LIN {X 0,Y 358.84,Z 342.917,A -85,B 0,C 180,E1 -13392.769,E2 -13392.769} C_VEL
LIN {X 0,Y 357.605,Z 354.158,A -85,B 0,C 180,E1 -13394.029,E2 -13394.029} C_VEL
LIN {X 0,Y 356.532,Z 364.122,A -85,B 0,C 180,E1 -13395.444,E2 -13395.444} C_VEL
LIN {X 0,Y 355.516,Z 373.786,A -85,B 0,C 180,E1 -13397.15,E2 -13397.15} C_VEL
LIN {X 0,Y 354.57,Z 381.475,A -85,B 0,C 180,E1 -13398.857,E2 -13398.857} C_VEL
LIN {X 0,Y 353.885,Z 388.571,A -85,B 0,C 180,E1 -13400.858,E2 -13400.858} C_VEL
LIN {X 0,Y 353.515,Z 393.294,A -85,B 0,C 180,E1 -13402.575,E2 -13402.575} C_VEL
LIN {X 0,Y 353.31,Z 396.903,A -85,B 0,C 180,E1 -13404.292,E2 -13404.292} C_VEL
LIN {X 0,Y 353.278,Z 398.766,A -85,B 0,C 180,E1 -13405.436,E2 -13405.436} C_VEL
LIN {X 0,Y 353.222,Z 400.162,A -85,B 0,C 180,E1 -13406.578,E2 -13406.578} C_VEL
LIN {X 0,Y 353.216,Z 401.767,A -85,B 0,C 180,E1 -13408.86,E2 -13408.86} C_VEL
LIN {X 0,Y 353.262,Z 401.983,A -85,B 0,C 180,E1 -13410,E2 -13410} C_VEL
LIN {X 0,Y 353.216,Z 401.762,A -85,B 0,C 180,E1 -13411.14,E2 -13411.14} C_VEL
LIN {X 0,Y 353.219,Z 400.153,A -85,B 0,C 180,E1 -13413.422,E2 -13413.422} C_VEL
LIN {X 0,Y 353.263,Z 398.752,A -85,B 0,C 180,E1 -13414.564,E2 -13414.564} C_VEL
LIN {X 0,Y 353.278,Z 396.508,A -85,B 0,C 180,E1 -13415.908,E2 -13415.908} C_VEL
LIN {X 0,Y 353.615,Z 391.828,A -85,B 0,C 180,E1 -13417.997,E2 -13417.997} C_VEL
LIN {X 0,Y 354.162,Z 385.708,A -85,B 0,C 180,E1 -13419.999,E2 -13419.999} C_VEL
LIN {X 0,Y 354.828,Z 379.025,A -85,B 0,C 180,E1 -13421.714,E2 -13421.714} C_VEL
LIN {X 0,Y 355.87,Z 370.739,A -85,B 0,C 180,E1 -13423.418,E2 -13423.418} C_VEL
LIN {X 0,Y 356.797,Z 362.241,A -85,B 0,C 180,E1 -13424.837,E2 -13424.837} C_VEL
LIN {X 0,Y 357.874,Z 351.742,A -85,B 0,C 180,E1 -13426.251,E2 -13426.251} C_VEL
LIN {X 0,Y 359.111,Z 339.929,A -85,B 0,C 180,E1 -13427.511,E2 -13427.511} C_VEL
LIN {X 0,Y 359.835,Z 331.742,A -85,B 0,C 180,E1 -13428.21,E2 -13428.21} C_VEL
LIN {X 0,Y 358.663,Z 320.559,A -85,B 0,C 180,E1 -13429.087,E2 -13429.087} C_VEL
LIN {X 0,Y 356.717,Z 308.163,A -85,B 0,C 180,E1 -13429.872,E2 -13429.872} C_VEL
LIN {X 0,Y 354.087,Z 295.342,A -85,B 0,C 180,E1 -13430.496,E2 -13430.496} C_VEL
LIN {X 0,Y 354.506,Z 288.95,A -85,B 0,C 180,E1 -13434.225,E2 -13434.225} C_VEL
LIN {X 0,Y 355.003,Z 283.001,A -85,B 0,C 180,E1 -13437.725,E2 -13437.725} C_VEL
LIN {X 0,Y 355.574,Z 277.671,A -85,B 0,C 180,E1 -13440.924,E2 -13440.924} C_VEL
LIN {X 0,Y 356.224,Z 271.24,A -85,B 0,C 180,E1 -13444.9,E2 -13444.9} C_VEL
LIN {X 0,Y 356.056,Z 266.77,A -85,B 0,C 180,E1 -13447.857,E2 -13447.857} C_VEL
LIN {X 0,Y 355.303,Z 261.976,A -85,B 0,C 180,E1 -13451.266,E2 -13451.266} C_VEL
LIN {X 0,Y 354.831,Z 259.291,A -85,B 0,C 180,E1 -13453.339,E2 -13453.339} C_VEL
LIN {X 0,Y 354.786,Z 259.29,A -85,B 0,C 180,E1 -13457.133,E2 -13457.133} C_VEL
LIN {X 0,Y 354.785,Z 259.294,A -85,B 0,C 180,E1 -13460.662,E2 -13460.662} C_VEL
LIN {X 0,Y 354.822,Z 259.288,A -85,B 0,C 180,E1 -13464.301,E2 -13464.301} C_VEL
LIN {X 0,Y 354.788,Z 259.289,A -85,B 0,C 180,E1 -13467.667,E2 -13467.667} C_VEL
LIN {X 0,Y 354.802,Z 259.287,A -85,B 0,C 180,E1 -13471.615,E2 -13471.615} C_VEL
LIN {X 0,Y 354.806,Z 259.286,A -85,B 0,C 180,E1 -13475.42,E2 -13475.42} C_VEL
LIN {X 0,Y 354.828,Z 259.283,A -85,B 0,C 180,E1 -13479.113,E2 -13479.113} C_VEL
LIN {X 0,Y 354.9,Z 259.274,A -85,B 0,C 180,E1 -13482.72,E2 -13482.72} C_VEL
LIN {X 0,Y 354.953,Z 259.269,A -85,B 0,C 180,E1 -13486.255,E2 -13486.255} C_VEL
LIN {X 0,Y 354.956,Z 259.271,A -85,B 0,C 180,E1 -13489.735,E2 -13489.735} C_VEL
LIN {X 0,Y 355.113,Z 259.25,A -85,B 0,C 180,E1 -13493.18,E2 -13493.18} C_VEL
LIN {X 0,Y 355.245,Z 259.233,A -85,B 0,C 180,E1 -13497.732,E2 -13497.732} C_VEL
LIN {X 0,Y 355.353,Z 259.218,A -85,B 0,C 180,E1 -13500,E2 -13500} C_VEL
LIN {X 0,Y 355.232,Z 259.233,A -85,B 0,C 180,E1 -13502.268,E2 -13502.268} C_VEL
LIN {X 0,Y 355.107,Z 259.252,A -85,B 0,C 180,E1 -13506.82,E2 -13506.82} C_VEL
LIN {X 0,Y 354.958,Z 259.268,A -85,B 0,C 180,E1 -13510.265,E2 -13510.265} C_VEL
LIN {X 0,Y 354.944,Z 259.269,A -85,B 0,C 180,E1 -13514.019,E2 -13514.019} C_VEL
LIN {X 0,Y 354.891,Z 259.276,A -85,B 0,C 180,E1 -13518.092,E2 -13518.092} C_VEL
LIN {X 0,Y 354.817,Z 259.287,A -85,B 0,C 180,E1 -13522.107,E2 -13522.107} C_VEL
LIN {X 0,Y 354.9,Z 259.275,A -85,B 0,C 180,E1 -13525.828,E2 -13525.828} C_VEL
LIN {X 0,Y 354.855,Z 259.281,A -85,B 0,C 180,E1 -13529.679,E2 -13529.679} C_VEL
LIN {X 0,Y 354.807,Z 259.288,A -85,B 0,C 180,E1 -13533.702,E2 -13533.702} C_VEL
LIN {X 0,Y 354.796,Z 259.289,A -85,B 0,C 180,E1 -13536.46,E2 -13536.46} C_VEL
LIN {X 0,Y 354.825,Z 259.285,A -85,B 0,C 180,E1 -13539.424,E2 -13539.424} C_VEL
LIN {X 0,Y 354.787,Z 259.288,A -85,B 0,C 180,E1 -13542.867,E2 -13542.867} C_VEL
LIN {X 0,Y 354.763,Z 259.293,A -85,B 0,C 180,E1 -13546.103,E2 -13546.103} C_VEL
LIN {X 0,Y 354.763,Z 259.294,A -85,B 0,C 180,E1 -13549.176,E2 -13549.176} C_VEL
LIN {X 0,Y 354.781,Z 259.293,A -85,B 0,C 180,E1 -13552.408,E2 -13552.408} C_VEL
LIN {X 0,Y 354.752,Z 259.395,A -85,B 0,C 180,E1 -13553.535,E2 -13553.535} C_VEL
LIN {X 0,Y 354.712,Z 262.351,A -85,B 0,C 180,E1 -13556.321,E2 -13556.321} C_VEL
LIN {X 0,Y 354.545,Z 265.242,A -85,B 0,C 180,E1 -13558.977,E2 -13558.977} C_VEL
LIN {X 0,Y 354.359,Z 268.174,A -85,B 0,C 180,E1 -13561.576,E2 -13561.576} C_VEL
LIN {X 0,Y 354.181,Z 271.128,A -85,B 0,C 180,E1 -13564.116,E2 -13564.116} C_VEL
LIN {X 0,Y 354.025,Z 274.086,A -85,B 0,C 180,E1 -13566.607,E2 -13566.607} C_VEL
LIN {X 0,Y 353.896,Z 277.951,A -85,B 0,C 180,E1 -13569.582,E2 -13569.582} C_VEL
LIN {X 0,Y 357.36,Z 291.296,A -85,B 0,C 180,E1 -13570.311,E2 -13570.311} C_VEL
LIN {X 0,Y 360.034,Z 303.79,A -85,B 0,C 180,E1 -13571.188,E2 -13571.188} C_VEL
LIN {X 0,Y 360.75,Z 309.963,A -85,B 0,C 180,E1 -13571.676,E2 -13571.676} C_VEL
LIN {X 0,Y 359.733,Z 321.615,A -85,B 0,C 180,E1 -13572.666,E2 -13572.666} C_VEL
LIN {X 0,Y 358.763,Z 332.231,A -85,B 0,C 180,E1 -13573.817,E2 -13573.817} C_VEL
LIN {X 0,Y 357.607,Z 342.508,A -85,B 0,C 180,E1 -13575.198,E2 -13575.198} C_VEL
LIN {X 0,Y 356.595,Z 351.002,A -85,B 0,C 180,E1 -13576.61,E2 -13576.61} C_VEL
LIN {X 0,Y 355.567,Z 359.255,A -85,B 0,C 180,E1 -13578.311,E2 -13578.311} C_VEL
LIN {X 0,Y 354.765,Z 365.902,A -85,B 0,C 180,E1 -13580.018,E2 -13580.018} C_VEL
LIN {X 0,Y 354.082,Z 371.99,A -85,B 0,C 180,E1 -13582.014,E2 -13582.014} C_VEL
LIN {X 0,Y 353.808,Z 375.059,A -85,B 0,C 180,E1 -13583.314,E2 -13583.314} C_VEL
LIN {X 0,Y 353.494,Z 378.859,A -85,B 0,C 180,E1 -13585.439,E2 -13585.439} C_VEL
LIN {X 0,Y 353.335,Z 380.259,A -85,B 0,C 180,E1 -13586.579,E2 -13586.579} C_VEL
LIN {X 0,Y 353.256,Z 381.864,A -85,B 0,C 180,E1 -13588.86,E2 -13588.86} C_VEL
LIN {X 0,Y 353.265,Z 382.096,A -85,B 0,C 180,E1 -13590,E2 -13590} C_VEL
LIN {X 0,Y 353.256,Z 381.907,A -85,B 0,C 180,E1 -13591.14,E2 -13591.14} C_VEL
LIN {X 0,Y 353.332,Z 380.356,A -85,B 0,C 180,E1 -13593.421,E2 -13593.421} C_VEL
LIN {X 0,Y 353.486,Z 378.999,A -85,B 0,C 180,E1 -13594.562,E2 -13594.562} C_VEL
LIN {X 0,Y 353.738,Z 376.181,A -85,B 0,C 180,E1 -13596.247,E2 -13596.247} C_VEL
LIN {X 0,Y 354.088,Z 372.247,A -85,B 0,C 180,E1 -13597.986,E2 -13597.986} C_VEL
LIN {X 0,Y 354.62,Z 367.232,A -85,B 0,C 180,E1 -13599.698,E2 -13599.698} C_VEL
LIN {X 0,Y 355.366,Z 360.917,A -85,B 0,C 180,E1 -13601.407,E2 -13601.407} C_VEL
LIN {X 0,Y 356.347,Z 353.01,A -85,B 0,C 180,E1 -13603.109,E2 -13603.109} C_VEL
LIN {X 0,Y 357.578,Z 343.172,A -85,B 0,C 180,E1 -13604.804,E2 -13604.804} C_VEL
LIN {X 0,Y 358.681,Z 332.659,A -85,B 0,C 180,E1 -13606.237,E2 -13606.237} C_VEL
LIN {X 0,Y 359.616,Z 322.621,A -85,B 0,C 180,E1 -13607.34,E2 -13607.34} C_VEL
LIN {X 0,Y 360.748,Z 310.987,A -85,B 0,C 180,E1 -13608.346,E2 -13608.346} C_VEL
LIN {X 0,Y 360.615,Z 307.38,A -85,B 0,C 180,E1 -13608.628,E2 -13608.628} C_VEL
LIN {X 0,Y 358.493,Z 296.304,A -85,B 0,C 180,E1 -13609.468,E2 -13609.468} C_VEL
LIN {X 0,Y 355.47,Z 283.821,A -85,B 0,C 180,E1 -13610.233,E2 -13610.233} C_VEL
LIN {X 0,Y 353.884,Z 277.728,A -85,B 0,C 180,E1 -13610.556,E2 -13610.556} C_VEL
LIN {X 0,Y 354.106,Z 272.742,A -85,B 0,C 180,E1 -13614.632,E2 -13614.632} C_VEL
LIN {X 0,Y 354.281,Z 269.783,A -85,B 0,C 180,E1 -13617.146,E2 -13617.146} C_VEL
LIN {X 0,Y 354.421,Z 266.827,A -85,B 0,C 180,E1 -13619.719,E2 -13619.719} C_VEL
LIN {X 0,Y 354.596,Z 263.203,A -85,B 0,C 180,E1 -13622.991,E2 -13622.991} C_VEL
LIN {X 0,Y 354.759,Z 260.333,A -85,B 0,C 180,E1 -13625.685,E2 -13625.685} C_VEL
LIN {X 0,Y 354.736,Z 259.52,A -85,B 0,C 180,E1 -13626.467,E2 -13626.467} C_VEL
LIN {X 0,Y 354.774,Z 259.292,A -85,B 0,C 180,E1 -13627.861,E2 -13627.861} C_VEL
LIN {X 0,Y 354.124,Z 259.375,A -85,B 0,C 180,E1 -13628.807,E2 -13628.807} C_VEL
LIN {X 0,Y 351.253,Z 259.732,A -85,B 0,C 180,E1 -13630.347,E2 -13630.347} C_VEL
LIN {X 0,Y 348.817,Z 260.031,A -85,B 0,C 180,E1 -13631.593,E2 -13631.593} C_VEL
LIN {X 0,Y 347.784,Z 260.165,A -85,B 0,C 180,E1 -13632.557,E2 -13632.557} C_VEL
LIN {X 0,Y 347.707,Z 260.167,A -85,B 0,C 180,E1 -13632.884,E2 -13632.884} C_VEL
LIN {X 0,Y 347.727,Z 260.17,A -85,B 0,C 180,E1 -13636.686,E2 -13636.686} C_VEL
LIN {X 0,Y 347.748,Z 260.171,A -85,B 0,C 180,E1 -13640.173,E2 -13640.173} C_VEL
LIN {X 0,Y 347.763,Z 260.164,A -85,B 0,C 180,E1 -13642.679,E2 -13642.679} C_VEL
LIN {X 0,Y 347.751,Z 260.17,A -85,B 0,C 180,E1 -13645.956,E2 -13645.956} C_VEL
LIN {X 0,Y 347.766,Z 260.166,A -85,B 0,C 180,E1 -13649.654,E2 -13649.654} C_VEL
LIN {X 0,Y 347.854,Z 260.151,A -85,B 0,C 180,E1 -13652.745,E2 -13652.745} C_VEL
LIN {X 0,Y 347.787,Z 260.161,A -85,B 0,C 180,E1 -13656.162,E2 -13656.162} C_VEL
LIN {X 0,Y 347.802,Z 260.16,A -85,B 0,C 180,E1 -13659.909,E2 -13659.909} C_VEL
LIN {X 0,Y 347.834,Z 260.158,A -85,B 0,C 180,E1 -13663.568,E2 -13663.568} C_VEL
LIN {X 0,Y 347.893,Z 260.152,A -85,B 0,C 180,E1 -13667.161,E2 -13667.161} C_VEL
LIN {X 0,Y 347.938,Z 260.143,A -85,B 0,C 180,E1 -13670.701,E2 -13670.701} C_VEL
LIN {X 0,Y 348.076,Z 260.13,A -85,B 0,C 180,E1 -13673.042,E2 -13673.042} C_VEL
LIN {X 0,Y 348.195,Z 260.109,A -85,B 0,C 180,E1 -13677.686,E2 -13677.686} C_VEL
LIN {X 0,Y 348.148,Z 260.117,A -85,B 0,C 180,E1 -13681.157,E2 -13681.157} C_VEL
LIN {X 0,Y 348.209,Z 260.11,A -85,B 0,C 180,E1 -13682.313,E2 -13682.313} C_VEL
LIN {X 0,Y 348.08,Z 260.126,A -85,B 0,C 180,E1 -13686.958,E2 -13686.958} C_VEL
LIN {X 0,Y 347.894,Z 260.152,A -85,B 0,C 180,E1 -13690.475,E2 -13690.475} C_VEL
LIN {X 0,Y 347.901,Z 260.15,A -85,B 0,C 180,E1 -13694.15,E2 -13694.15} C_VEL
LIN {X 0,Y 347.894,Z 260.151,A -85,B 0,C 180,E1 -13698.29,E2 -13698.29} C_VEL
LIN {X 0,Y 347.769,Z 260.164,A -85,B 0,C 180,E1 -13701.626,E2 -13701.626} C_VEL
LIN {X 0,Y 347.743,Z 260.166,A -85,B 0,C 180,E1 -13705.114,E2 -13705.114} C_VEL
LIN {X 0,Y 347.74,Z 260.17,A -85,B 0,C 180,E1 -13707.7,E2 -13707.7} C_VEL
LIN {X 0,Y 347.743,Z 260.167,A -85,B 0,C 180,E1 -13710.349,E2 -13710.349} C_VEL
LIN {X 0,Y 347.75,Z 260.167,A -85,B 0,C 180,E1 -13714.044,E2 -13714.044} C_VEL
LIN {X 0,Y 347.758,Z 260.168,A -85,B 0,C 180,E1 -13717.321,E2 -13717.321} C_VEL
LIN {X 0,Y 347.742,Z 260.169,A -85,B 0,C 180,E1 -13721.601,E2 -13721.601} C_VEL
LIN {X 0,Y 347.707,Z 260.175,A -85,B 0,C 180,E1 -13725.027,E2 -13725.027} C_VEL
LIN {X 0,Y 347.797,Z 260.363,A -85,B 0,C 180,E1 -13726.503,E2 -13726.503} C_VEL
LIN {X 0,Y 348.598,Z 264.999,A -85,B 0,C 180,E1 -13730.006,E2 -13730.006} C_VEL
LIN {X 0,Y 349.207,Z 269.003,A -85,B 0,C 180,E1 -13732.859,E2 -13732.859} C_VEL
LIN {X 0,Y 349.145,Z 273.279,A -85,B 0,C 180,E1 -13735.693,E2 -13735.693} C_VEL
LIN {X 0,Y 348.401,Z 279.687,A -85,B 0,C 180,E1 -13739.715,E2 -13739.715} C_VEL
LIN {X 0,Y 347.715,Z 286.034,A -85,B 0,C 180,E1 -13743.598,E2 -13743.598} C_VEL
LIN {X 0,Y 347.277,Z 292.338,A -85,B 0,C 180,E1 -13747.386,E2 -13747.386} C_VEL
LIN {X 0,Y 347.056,Z 295.141,A -85,B 0,C 180,E1 -13749.05,E2 -13749.05} C_VEL
LIN {X 0,Y 350.069,Z 309.551,A -85,B 0,C 180,E1 -13749.797,E2 -13749.797} C_VEL
LIN {X 0,Y 351.916,Z 321.47,A -85,B 0,C 180,E1 -13750.592,E2 -13750.592} C_VEL
LIN {X 0,Y 353.017,Z 333.482,A -85,B 0,C 180,E1 -13751.576,E2 -13751.576} C_VEL
LIN {X 0,Y 351.882,Z 344.141,A -85,B 0,C 180,E1 -13752.567,E2 -13752.567} C_VEL
LIN {X 0,Y 350.633,Z 355.073,A -85,B 0,C 180,E1 -13753.858,E2 -13753.858} C_VEL
LIN {X 0,Y 349.631,Z 363.923,A -85,B 0,C 180,E1 -13755.15,E2 -13755.15} C_VEL
LIN {X 0,Y 348.555,Z 373.587,A -85,B 0,C 180,E1 -13756.889,E2 -13756.889} C_VEL
LIN {X 0,Y 347.55,Z 381.275,A -85,B 0,C 180,E1 -13758.629,E2 -13758.629} C_VEL
LIN {X 0,Y 346.857,Z 388.372,A -85,B 0,C 180,E1 -13760.671,E2 -13760.671} C_VEL
LIN {X 0,Y 346.465,Z 393.095,A -85,B 0,C 180,E1 -13762.423,E2 -13762.423} C_VEL
LIN {X 0,Y 346.23,Z 396.704,A -85,B 0,C 180,E1 -13764.175,E2 -13764.175} C_VEL
LIN {X 0,Y 346.176,Z 398.566,A -85,B 0,C 180,E1 -13765.342,E2 -13765.342} C_VEL
LIN {X 0,Y 346.146,Z 399.963,A -85,B 0,C 180,E1 -13766.508,E2 -13766.508} C_VEL
LIN {X 0,Y 346.116,Z 401.567,A -85,B 0,C 180,E1 -13768.836,E2 -13768.836} C_VEL
LIN {X 0,Y 346.164,Z 401.783,A -85,B 0,C 180,E1 -13770,E2 -13770} C_VEL
LIN {X 0,Y 346.116,Z 401.562,A -85,B 0,C 180,E1 -13771.163,E2 -13771.163} C_VEL
LIN {X 0,Y 346.142,Z 399.953,A -85,B 0,C 180,E1 -13773.492,E2 -13773.492} C_VEL
LIN {X 0,Y 346.16,Z 398.551,A -85,B 0,C 180,E1 -13774.658,E2 -13774.658} C_VEL
LIN {X 0,Y 346.241,Z 395.608,A -85,B 0,C 180,E1 -13776.409,E2 -13776.409} C_VEL
LIN {X 0,Y 346.555,Z 391.626,A -85,B 0,C 180,E1 -13778.161,E2 -13778.161} C_VEL
LIN {X 0,Y 347.136,Z 385.506,A -85,B 0,C 180,E1 -13780.204,E2 -13780.204} C_VEL
LIN {X 0,Y 347.825,Z 378.821,A -85,B 0,C 180,E1 -13781.953,E2 -13781.953} C_VEL
LIN {X 0,Y 348.941,Z 370.536,A -85,B 0,C 180,E1 -13783.689,E2 -13783.689} C_VEL
LIN {X 0,Y 350.023,Z 360.981,A -85,B 0,C 180,E1 -13785.292,E2 -13785.292} C_VEL
LIN {X 0,Y 351.191,Z 350.362,A -85,B 0,C 180,E1 -13786.719,E2 -13786.719} C_VEL
LIN {X 0,Y 352.35,Z 339.725,A -85,B 0,C 180,E1 -13787.859,E2 -13787.859} C_VEL
LIN {X 0,Y 352.914,Z 331.531,A -85,B 0,C 180,E1 -13788.58,E2 -13788.58} C_VEL
LIN {X 0,Y 351.632,Z 319.183,A -85,B 0,C 180,E1 -13789.561,E2 -13789.561} C_VEL
LIN {X 0,Y 349.365,Z 306.037,A -85,B 0,C 180,E1 -13790.389,E2 -13790.389} C_VEL
LIN {X 0,Y 347.068,Z 295.148,A -85,B 0,C 180,E1 -13790.929,E2 -13790.929} C_VEL
LIN {X 0,Y 347.489,Z 289.211,A -85,B 0,C 180,E1 -13794.476,E2 -13794.476} C_VEL
LIN {X 0,Y 348.025,Z 282.822,A -85,B 0,C 180,E1 -13798.331,E2 -13798.331} C_VEL
LIN {X 0,Y 348.626,Z 277.509,A -85,B 0,C 180,E1 -13801.61,E2 -13801.61} C_VEL
LIN {X 0,Y 349.202,Z 272.159,A -85,B 0,C 180,E1 -13805,E2 -13805} C_VEL
LIN {X 0,Y 349.176,Z 268.964,A -85,B 0,C 180,E1 -13807.144,E2 -13807.144} C_VEL
LIN {X 0,Y 348.54,Z 264.698,A -85,B 0,C 180,E1 -13810.184,E2 -13810.184} C_VEL
LIN {X 0,Y 347.779,Z 260.167,A -85,B 0,C 180,E1 -13813.699,E2 -13813.699} C_VEL
LIN {X 0,Y 347.725,Z 260.174,A -85,B 0,C 180,E1 -13816.686,E2 -13816.686} C_VEL
LIN {X 0,Y 347.701,Z 260.174,A -85,B 0,C 180,E1 -13820.182,E2 -13820.182} C_VEL
LIN {X 0,Y 347.757,Z 260.168,A -85,B 0,C 180,E1 -13822.678,E2 -13822.678} C_VEL
LIN {X 0,Y 347.749,Z 260.167,A -85,B 0,C 180,E1 -13825.956,E2 -13825.956} C_VEL
LIN {X 0,Y 347.742,Z 260.167,A -85,B 0,C 180,E1 -13829.651,E2 -13829.651} C_VEL
LIN {X 0,Y 347.747,Z 260.167,A -85,B 0,C 180,E1 -13833.601,E2 -13833.601} C_VEL
LIN {X 0,Y 347.749,Z 260.17,A -85,B 0,C 180,E1 -13836.159,E2 -13836.159} C_VEL
LIN {X 0,Y 347.813,Z 260.163,A -85,B 0,C 180,E1 -13839.909,E2 -13839.909} C_VEL
LIN {X 0,Y 347.868,Z 260.151,A -85,B 0,C 180,E1 -13842.359,E2 -13842.359} C_VEL
LIN {X 0,Y 347.899,Z 260.149,A -85,B 0,C 180,E1 -13845.971,E2 -13845.971} C_VEL
LIN {X 0,Y 347.897,Z 260.152,A -85,B 0,C 180,E1 -13849.525,E2 -13849.525} C_VEL
LIN {X 0,Y 348.079,Z 260.125,A -85,B 0,C 180,E1 -13853.042,E2 -13853.042} C_VEL
LIN {X 0,Y 348.207,Z 260.11,A -85,B 0,C 180,E1 -13857.687,E2 -13857.687} C_VEL
LIN {X 0,Y 348.304,Z 260.096,A -85,B 0,C 180,E1 -13860,E2 -13860} C_VEL
LIN {X 0,Y 348.193,Z 260.109,A -85,B 0,C 180,E1 -13862.314,E2 -13862.314} C_VEL
LIN {X 0,Y 348.074,Z 260.13,A -85,B 0,C 180,E1 -13866.958,E2 -13866.958} C_VEL
LIN {X 0,Y 347.899,Z 260.148,A -85,B 0,C 180,E1 -13870.475,E2 -13870.475} C_VEL
LIN {X 0,Y 347.9,Z 260.147,A -85,B 0,C 180,E1 -13874.15,E2 -13874.15} C_VEL
LIN {X 0,Y 347.83,Z 260.157,A -85,B 0,C 180,E1 -13878.259,E2 -13878.259} C_VEL
LIN {X 0,Y 347.769,Z 260.162,A -85,B 0,C 180,E1 -13881.626,E2 -13881.626} C_VEL
LIN {X 0,Y 347.813,Z 260.157,A -85,B 0,C 180,E1 -13885.109,E2 -13885.109} C_VEL
LIN {X 0,Y 347.812,Z 260.158,A -85,B 0,C 180,E1 -13887.694,E2 -13887.694} C_VEL
LIN {X 0,Y 347.765,Z 260.167,A -85,B 0,C 180,E1 -13890.347,E2 -13890.347} C_VEL
LIN {X 0,Y 347.744,Z 260.168,A -85,B 0,C 180,E1 -13894.464,E2 -13894.464} C_VEL
LIN {X 0,Y 347.772,Z 260.167,A -85,B 0,C 180,E1 -13897.988,E2 -13897.988} C_VEL
LIN {X 0,Y 347.749,Z 260.17,A -85,B 0,C 180,E1 -13901.831,E2 -13901.831} C_VEL
LIN {X 0,Y 347.703,Z 260.171,A -85,B 0,C 180,E1 -13905.027,E2 -13905.027} C_VEL
LIN {X 0,Y 347.738,Z 260.167,A -85,B 0,C 180,E1 -13908.4,E2 -13908.4} C_VEL
LIN {X 0,Y 347.752,Z 260.168,A -85,B 0,C 180,E1 -13912.016,E2 -13912.016} C_VEL
LIN {X 0,Y 347.734,Z 260.173,A -85,B 0,C 180,E1 -13912.676,E2 -13912.676} C_VEL
LIN {X 0,Y 347.741,Z 261.014,A -85,B 0,C 180,E1 -13914.119,E2 -13914.119} C_VEL
LIN {X 0,Y 347.617,Z 263.942,A -85,B 0,C 180,E1 -13916.915,E2 -13916.915} C_VEL
LIN {X 0,Y 347.392,Z 267.79,A -85,B 0,C 180,E1 -13920.45,E2 -13920.45} C_VEL
LIN {X 0,Y 347.189,Z 271.305,A -85,B 0,C 180,E1 -13923.555,E2 -13923.555} C_VEL
LIN {X 0,Y 347.032,Z 274.276,A -85,B 0,C 180,E1 -13926.107,E2 -13926.107} C_VEL
LIN {X 0,Y 346.827,Z 278.008,A -85,B 0,C 180,E1 -13929.141,E2 -13929.141} C_VEL
LIN {X 0,Y 350.344,Z 291.183,A -85,B 0,C 180,E1 -13929.883,E2 -13929.883} C_VEL
LIN {X 0,Y 353.068,Z 304.005,A -85,B 0,C 180,E1 -13930.803,E2 -13930.803} C_VEL
LIN {X 0,Y 354.017,Z 310.29,A -85,B 0,C 180,E1 -13931.324,E2 -13931.324} C_VEL
LIN {X 0,Y 352.963,Z 321.82,A -85,B 0,C 180,E1 -13932.323,E2 -13932.323} C_VEL
LIN {X 0,Y 351.878,Z 333.196,A -85,B 0,C 180,E1 -13933.589,E2 -13933.589} C_VEL
LIN {X 0,Y 350.756,Z 342.711,A -85,B 0,C 180,E1 -13934.902,E2 -13934.902} C_VEL
LIN {X 0,Y 349.685,Z 351.205,A -85,B 0,C 180,E1 -13936.341,E2 -13936.341} C_VEL
LIN {X 0,Y 348.625,Z 359.457,A -85,B 0,C 180,E1 -13938.075,E2 -13938.075} C_VEL
LIN {X 0,Y 347.775,Z 366.103,A -85,B 0,C 180,E1 -13939.815,E2 -13939.815} C_VEL
LIN {X 0,Y 347.045,Z 372.191,A -85,B 0,C 180,E1 -13941.851,E2 -13941.851} C_VEL
LIN {X 0,Y 346.731,Z 375.553,A -85,B 0,C 180,E1 -13943.315,E2 -13943.315} C_VEL
LIN {X 0,Y 346.436,Z 379.059,A -85,B 0,C 180,E1 -13945.346,E2 -13945.346} C_VEL
LIN {X 0,Y 346.26,Z 380.459,A -85,B 0,C 180,E1 -13946.509,E2 -13946.509} C_VEL
LIN {X 0,Y 346.159,Z 382.064,A -85,B 0,C 180,E1 -13948.837,E2 -13948.837} C_VEL
LIN {X 0,Y 346.168,Z 382.296,A -85,B 0,C 180,E1 -13950,E2 -13950} C_VEL
LIN {X 0,Y 346.159,Z 382.106,A -85,B 0,C 180,E1 -13951.163,E2 -13951.163} C_VEL
LIN {X 0,Y 346.257,Z 380.555,A -85,B 0,C 180,E1 -13953.491,E2 -13953.491} C_VEL
LIN {X 0,Y 346.428,Z 379.197,A -85,B 0,C 180,E1 -13954.655,E2 -13954.655} C_VEL
LIN {X 0,Y 346.791,Z 375.591,A -85,B 0,C 180,E1 -13956.769,E2 -13956.769} C_VEL
LIN {X 0,Y 347.221,Z 370.888,A -85,B 0,C 180,E1 -13958.732,E2 -13958.732} C_VEL
LIN {X 0,Y 347.997,Z 364.451,A -85,B 0,C 180,E1 -13960.767,E2 -13960.767} C_VEL
LIN {X 0,Y 348.869,Z 357.377,A -85,B 0,C 180,E1 -13962.507,E2 -13962.507} C_VEL
LIN {X 0,Y 350.055,Z 348.558,A -85,B 0,C 180,E1 -13964.238,E2 -13964.238} C_VEL
LIN {X 0,Y 351.182,Z 339.619,A -85,B 0,C 180,E1 -13965.657,E2 -13965.657} C_VEL
LIN {X 0,Y 352.19,Z 329.868,A -85,B 0,C 180,E1 -13966.924,E2 -13966.924} C_VEL
LIN {X 0,Y 353.203,Z 319.914,A -85,B 0,C 180,E1 -13967.964,E2 -13967.964} C_VEL
LIN {X 0,Y 354.051,Z 310.239,A -85,B 0,C 180,E1 -13968.783,E2 -13968.783} C_VEL
LIN {X 0,Y 352.005,Z 298.839,A -85,B 0,C 180,E1 -13969.704,E2 -13969.704} C_VEL
LIN {X 0,Y 349.157,Z 286.605,A -85,B 0,C 180,E1 -13970.506,E2 -13970.506} C_VEL
LIN {X 0,Y 346.826,Z 277.922,A -85,B 0,C 180,E1 -13971.003,E2 -13971.003} C_VEL
LIN {X 0,Y 347.036,Z 273.921,A -85,B 0,C 180,E1 -13974.311,E2 -13974.311} C_VEL
LIN {X 0,Y 347.263,Z 269.965,A -85,B 0,C 180,E1 -13977.741,E2 -13977.741} C_VEL
LIN {X 0,Y 347.433,Z 266.995,A -85,B 0,C 180,E1 -13980.379,E2 -13980.379} C_VEL
LIN {X 0,Y 347.661,Z 263.079,A -85,B 0,C 180,E1 -13984.022,E2 -13984.022} C_VEL
LIN {X 0,Y 347.737,Z 260.956,A -85,B 0,C 180,E1 -13986.057,E2 -13986.057} C_VEL
LIN {X 0,Y 347.699,Z 260.175,A -85,B 0,C 180,E1 -13987.329,E2 -13987.329} C_VEL
LIN {X 0,Y 347.699,Z 260.174,A -85,B 0,C 180,E1 -13990.302,E2 -13990.302} C_VEL
LIN {X 0,Y 347.707,Z 260.167,A -85,B 0,C 180,E1 -13992.884,E2 -13992.884} C_VEL
LIN {X 0,Y 347.069,Z 260.251,A -85,B 0,C 180,E1 -13993.851,E2 -13993.851} C_VEL
LIN {X 0,Y 344.257,Z 260.607,A -85,B 0,C 180,E1 -13995.425,E2 -13995.425} C_VEL
LIN {X 0,Y 341.846,Z 260.907,A -85,B 0,C 180,E1 -13996.699,E2 -13996.699} C_VEL
LIN {X 0,Y 340.791,Z 261.036,A -85,B 0,C 180,E1 -13997.684,E2 -13997.684} C_VEL
LIN {X 0,Y 340.695,Z 261.046,A -85,B 0,C 180,E1 -13998.018,E2 -13998.018} C_VEL
LIN {X 0,Y 340.734,Z 261.041,A -85,B 0,C 180,E1 -14001.773,E2 -14001.773} C_VEL
LIN {X 0,Y 340.725,Z 261.042,A -85,B 0,C 180,E1 -14005.595,E2 -14005.595} C_VEL
LIN {X 0,Y 340.706,Z 261.042,A -85,B 0,C 180,E1 -14008.956,E2 -14008.956} C_VEL
LIN {X 0,Y 340.781,Z 261.033,A -85,B 0,C 180,E1 -14012.474,E2 -14012.474} C_VEL
LIN {X 0,Y 340.757,Z 261.041,A -85,B 0,C 180,E1 -14015.638,E2 -14015.638} C_VEL
LIN {X 0,Y 340.733,Z 261.044,A -85,B 0,C 180,E1 -14019.473,E2 -14019.473} C_VEL
LIN {X 0,Y 340.795,Z 261.032,A -85,B 0,C 180,E1 -14021.981,E2 -14021.981} C_VEL
LIN {X 0,Y 340.872,Z 261.024,A -85,B 0,C 180,E1 -14025.705,E2 -14025.705} C_VEL
LIN {X 0,Y 340.852,Z 261.029,A -85,B 0,C 180,E1 -14029.306,E2 -14029.306} C_VEL
LIN {X 0,Y 341.023,Z 261.007,A -85,B 0,C 180,E1 -14032.897,E2 -14032.897} C_VEL
LIN {X 0,Y 340.827,Z 261.03,A -85,B 0,C 180,E1 -14035.269,E2 -14035.269} C_VEL
LIN {X 0,Y 341.132,Z 260.99,A -85,B 0,C 180,E1 -14037.638,E2 -14037.638} C_VEL
LIN {X 0,Y 341.117,Z 260.993,A -85,B 0,C 180,E1 -14041.18,E2 -14041.18} C_VEL
LIN {X 0,Y 341.17,Z 260.987,A -85,B 0,C 180,E1 -14042.361,E2 -14042.361} C_VEL
LIN {X 0,Y 341.048,Z 261.001,A -85,B 0,C 180,E1 -14047.102,E2 -14047.102} C_VEL
LIN {X 0,Y 340.846,Z 261.028,A -85,B 0,C 180,E1 -14050.695,E2 -14050.695} C_VEL
LIN {X 0,Y 340.866,Z 261.028,A -85,B 0,C 180,E1 -14054.325,E2 -14054.325} C_VEL
LIN {X 0,Y 340.841,Z 261.028,A -85,B 0,C 180,E1 -14058.467,E2 -14058.467} C_VEL
LIN {X 0,Y 340.72,Z 261.044,A -85,B 0,C 180,E1 -14061.842,E2 -14061.842} C_VEL
LIN {X 0,Y 340.679,Z 261.049,A -85,B 0,C 180,E1 -14065.672,E2 -14065.672} C_VEL
LIN {X 0,Y 340.685,Z 261.046,A -85,B 0,C 180,E1 -14068.325,E2 -14068.325} C_VEL
LIN {X 0,Y 340.696,Z 261.044,A -85,B 0,C 180,E1 -14071.045,E2 -14071.045} C_VEL
LIN {X 0,Y 340.72,Z 261.044,A -85,B 0,C 180,E1 -14075.279,E2 -14075.279} C_VEL
LIN {X 0,Y 340.695,Z 261.044,A -85,B 0,C 180,E1 -14078.382,E2 -14078.382} C_VEL
LIN {X 0,Y 340.695,Z 261.045,A -85,B 0,C 180,E1 -14082.044,E2 -14082.044} C_VEL
LIN {X 0,Y 340.711,Z 261.115,A -85,B 0,C 180,E1 -14086.056,E2 -14086.056} C_VEL
LIN {X 0,Y 341.528,Z 265.666,A -85,B 0,C 180,E1 -14089.587,E2 -14089.587} C_VEL
LIN {X 0,Y 342.033,Z 268.865,A -85,B 0,C 180,E1 -14091.944,E2 -14091.944} C_VEL
LIN {X 0,Y 342.225,Z 272.054,A -85,B 0,C 180,E1 -14094.177,E2 -14094.177} C_VEL
LIN {X 0,Y 341.976,Z 275.259,A -85,B 0,C 180,E1 -14096.297,E2 -14096.297} C_VEL
LIN {X 0,Y 341.309,Z 280.827,A -85,B 0,C 180,E1 -14099.864,E2 -14099.864} C_VEL
LIN {X 0,Y 340.644,Z 286.911,A -85,B 0,C 180,E1 -14103.667,E2 -14103.667} C_VEL
LIN {X 0,Y 340.175,Z 293.187,A -85,B 0,C 180,E1 -14107.529,E2 -14107.529} C_VEL
LIN {X 0,Y 340.036,Z 294.938,A -85,B 0,C 180,E1 -14108.599,E2 -14108.599} C_VEL
LIN {X 0,Y 343.044,Z 309.043,A -85,B 0,C 180,E1 -14109.349,E2 -14109.349} C_VEL
LIN {X 0,Y 345.045,Z 321.68,A -85,B 0,C 180,E1 -14110.217,E2 -14110.217} C_VEL
LIN {X 0,Y 346.179,Z 333.285,A -85,B 0,C 180,E1 -14111.198,E2 -14111.198} C_VEL
LIN {X 0,Y 345.109,Z 343.945,A -85,B 0,C 180,E1 -14112.213,E2 -14112.213} C_VEL
LIN {X 0,Y 343.784,Z 354.943,A -85,B 0,C 180,E1 -14113.537,E2 -14113.537} C_VEL
LIN {X 0,Y 342.745,Z 363.725,A -85,B 0,C 180,E1 -14114.844,E2 -14114.844} C_VEL
LIN {X 0,Y 341.617,Z 373.388,A -85,B 0,C 180,E1 -14116.618,E2 -14116.618} C_VEL
LIN {X 0,Y 340.554,Z 381.076,A -85,B 0,C 180,E1 -14118.392,E2 -14118.392} C_VEL
LIN {X 0,Y 340.025,Z 386.351,A -85,B 0,C 180,E1 -14119.881,E2 -14119.881} C_VEL
LIN {X 0,Y 339.514,Z 391.461,A -85,B 0,C 180,E1 -14121.668,E2 -14121.668} C_VEL
LIN {X 0,Y 339.204,Z 395.431,A -85,B 0,C 180,E1 -14123.457,E2 -14123.457} C_VEL
LIN {X 0,Y 339.079,Z 398.366,A -85,B 0,C 180,E1 -14125.244,E2 -14125.244} C_VEL
LIN {X 0,Y 339.07,Z 399.764,A -85,B 0,C 180,E1 -14126.435,E2 -14126.435} C_VEL
LIN {X 0,Y 339.018,Z 401.368,A -85,B 0,C 180,E1 -14128.812,E2 -14128.812} C_VEL
LIN {X 0,Y 339.067,Z 401.583,A -85,B 0,C 180,E1 -14130,E2 -14130} C_VEL
LIN {X 0,Y 339.018,Z 401.362,A -85,B 0,C 180,E1 -14131.188,E2 -14131.188} C_VEL
LIN {X 0,Y 339.066,Z 399.753,A -85,B 0,C 180,E1 -14133.565,E2 -14133.565} C_VEL
LIN {X 0,Y 339.063,Z 398.35,A -85,B 0,C 180,E1 -14134.756,E2 -14134.756} C_VEL
LIN {X 0,Y 339.166,Z 395.405,A -85,B 0,C 180,E1 -14136.544,E2 -14136.544} C_VEL
LIN {X 0,Y 339.514,Z 391.425,A -85,B 0,C 180,E1 -14138.331,E2 -14138.331} C_VEL
LIN {X 0,Y 340.116,Z 385.304,A -85,B 0,C 180,E1 -14140.417,E2 -14140.417} C_VEL
LIN {X 0,Y 340.849,Z 378.619,A -85,B 0,C 180,E1 -14142.201,E2 -14142.201} C_VEL
LIN {X 0,Y 342.016,Z 370.333,A -85,B 0,C 180,E1 -14143.972,E2 -14143.972} C_VEL
LIN {X 0,Y 343.149,Z 360.752,A -85,B 0,C 180,E1 -14145.61,E2 -14145.61} C_VEL
LIN {X 0,Y 344.38,Z 350.158,A -85,B 0,C 180,E1 -14147.059,E2 -14147.059} C_VEL
LIN {X 0,Y 345.603,Z 339.521,A -85,B 0,C 180,E1 -14148.219,E2 -14148.219} C_VEL
LIN {X 0,Y 346.116,Z 333.099,A -85,B 0,C 180,E1 -14148.805,E2 -14148.805} C_VEL
LIN {X 0,Y 345.045,Z 321.908,A -85,B 0,C 180,E1 -14149.75,E2 -14149.75} C_VEL
LIN {X 0,Y 342.949,Z 308.971,A -85,B 0,C 180,E1 -14150.642,E2 -14150.642} C_VEL
LIN {X 0,Y 340.307,Z 296.664,A -85,B 0,C 180,E1 -14151.305,E2 -14151.305} C_VEL
LIN {X 0,Y 340.036,Z 294.935,A -85,B 0,C 180,E1 -14151.385,E2 -14151.385} C_VEL
LIN {X 0,Y 340.452,Z 289.491,A -85,B 0,C 180,E1 -14154.728,E2 -14154.728} C_VEL
LIN {X 0,Y 340.975,Z 283.706,A -85,B 0,C 180,E1 -14158.298,E2 -14158.298} C_VEL
LIN {X 0,Y 341.584,Z 278.412,A -85,B 0,C 180,E1 -14161.645,E2 -14161.645} C_VEL
LIN {X 0,Y 342.194,Z 273.071,A -85,B 0,C 180,E1 -14165.104,E2 -14165.104} C_VEL
LIN {X 0,Y 341.997,Z 268.801,A -85,B 0,C 180,E1 -14168.061,E2 -14168.061} C_VEL
LIN {X 0,Y 341.348,Z 264.549,A -85,B 0,C 180,E1 -14171.212,E2 -14171.212} C_VEL
LIN {X 0,Y 340.707,Z 261.048,A -85,B 0,C 180,E1 -14173.999,E2 -14173.999} C_VEL
LIN {X 0,Y 340.694,Z 261.044,A -85,B 0,C 180,E1 -14177.956,E2 -14177.956} C_VEL
LIN {X 0,Y 340.719,Z 261.041,A -85,B 0,C 180,E1 -14181.771,E2 -14181.771} C_VEL
LIN {X 0,Y 340.724,Z 261.041,A -85,B 0,C 180,E1 -14185.595,E2 -14185.595} C_VEL
LIN {X 0,Y 340.695,Z 261.045,A -85,B 0,C 180,E1 -14188.955,E2 -14188.955} C_VEL
LIN {X 0,Y 340.72,Z 261.041,A -85,B 0,C 180,E1 -14193.013,E2 -14193.013} C_VEL
LIN {X 0,Y 340.702,Z 261.043,A -85,B 0,C 180,E1 -14196.925,E2 -14196.925} C_VEL
LIN {X 0,Y 340.794,Z 261.031,A -85,B 0,C 180,E1 -14200.734,E2 -14200.734} C_VEL
LIN {X 0,Y 340.788,Z 261.033,A -85,B 0,C 180,E1 -14203.219,E2 -14203.219} C_VEL
LIN {X 0,Y 340.845,Z 261.025,A -85,B 0,C 180,E1 -14206.891,E2 -14206.891} C_VEL
LIN {X 0,Y 340.883,Z 261.02,A -85,B 0,C 180,E1 -14210.506,E2 -14210.506} C_VEL
LIN {X 0,Y 341.047,Z 261.001,A -85,B 0,C 180,E1 -14212.898,E2 -14212.898} C_VEL
LIN {X 0,Y 341.169,Z 260.987,A -85,B 0,C 180,E1 -14217.639,E2 -14217.639} C_VEL
LIN {X 0,Y 341.255,Z 260.974,A -85,B 0,C 180,E1 -14220,E2 -14220} C_VEL
LIN {X 0,Y 341.131,Z 260.989,A -85,B 0,C 180,E1 -14222.362,E2 -14222.362} C_VEL
LIN {X 0,Y 341.043,Z 261.005,A -85,B 0,C 180,E1 -14227.103,E2 -14227.103} C_VEL
LIN {X 0,Y 340.85,Z 261.028,A -85,B 0,C 180,E1 -14230.695,E2 -14230.695} C_VEL
LIN {X 0,Y 340.864,Z 261.024,A -85,B 0,C 180,E1 -14234.325,E2 -14234.325} C_VEL
LIN {X 0,Y 340.787,Z 261.036,A -85,B 0,C 180,E1 -14238.44,E2 -14238.44} C_VEL
LIN {X 0,Y 340.719,Z 261.041,A -85,B 0,C 180,E1 -14241.842,E2 -14241.842} C_VEL
LIN {X 0,Y 340.774,Z 261.034,A -85,B 0,C 180,E1 -14245.664,E2 -14245.664} C_VEL
LIN {X 0,Y 340.743,Z 261.043,A -85,B 0,C 180,E1 -14248.32,E2 -14248.32} C_VEL
LIN {X 0,Y 340.705,Z 261.042,A -85,B 0,C 180,E1 -14251.044,E2 -14251.044} C_VEL
LIN {X 0,Y 340.717,Z 261.041,A -85,B 0,C 180,E1 -14255.279,E2 -14255.279} C_VEL
LIN {X 0,Y 340.709,Z 261.044,A -85,B 0,C 180,E1 -14258.386,E2 -14258.386} C_VEL
LIN {X 0,Y 340.698,Z 261.047,A -85,B 0,C 180,E1 -14262.045,E2 -14262.045} C_VEL
LIN {X 0,Y 340.65,Z 261.05,A -85,B 0,C 180,E1 -14266.228,E2 -14266.228} C_VEL
LIN {X 0,Y 340.669,Z 261.048,A -85,B 0,C 180,E1 -14268.688,E2 -14268.688} C_VEL
LIN {X 0,Y 340.711,Z 261.046,A -85,B 0,C 180,E1 -14271.77,E2 -14271.77} C_VEL
LIN {X 0,Y 340.655,Z 261.164,A -85,B 0,C 180,E1 -14273.252,E2 -14273.252} C_VEL
LIN {X 0,Y 340.625,Z 264.115,A -85,B 0,C 180,E1 -14276.146,E2 -14276.146} C_VEL
LIN {X 0,Y 340.433,Z 267.043,A -85,B 0,C 180,E1 -14278.929,E2 -14278.929} C_VEL
LIN {X 0,Y 340.213,Z 271.146,A -85,B 0,C 180,E1 -14282.658,E2 -14282.658} C_VEL
LIN {X 0,Y 339.984,Z 274.469,A -85,B 0,C 180,E1 -14285.579,E2 -14285.579} C_VEL
LIN {X 0,Y 339.797,Z 278.158,A -85,B 0,C 180,E1 -14288.686,E2 -14288.686} C_VEL
LIN {X 0,Y 343.317,Z 291.304,A -85,B 0,C 180,E1 -14289.447,E2 -14289.447} C_VEL
LIN {X 0,Y 345.88,Z 303.126,A -85,B 0,C 180,E1 -14290.312,E2 -14290.312} C_VEL
LIN {X 0,Y 347.186,Z 310.646,A -85,B 0,C 180,E1 -14290.955,E2 -14290.955} C_VEL
LIN {X 0,Y 346.197,Z 322.025,A -85,B 0,C 180,E1 -14291.966,E2 -14291.966} C_VEL
LIN {X 0,Y 345.024,Z 333.711,A -85,B 0,C 180,E1 -14293.294,E2 -14293.294} C_VEL
LIN {X 0,Y 343.919,Z 342.914,A -85,B 0,C 180,E1 -14294.594,E2 -14294.594} C_VEL
LIN {X 0,Y 342.775,Z 351.408,A -85,B 0,C 180,E1 -14296.06,E2 -14296.06} C_VEL
LIN {X 0,Y 341.695,Z 359.659,A -85,B 0,C 180,E1 -14297.83,E2 -14297.83} C_VEL
LIN {X 0,Y 340.798,Z 366.305,A -85,B 0,C 180,E1 -14299.604,E2 -14299.604} C_VEL
LIN {X 0,Y 340.018,Z 372.392,A -85,B 0,C 180,E1 -14301.681,E2 -14301.681} C_VEL
LIN {X 0,Y 339.641,Z 376.084,A -85,B 0,C 180,E1 -14303.335,E2 -14303.335} C_VEL
LIN {X 0,Y 339.381,Z 379.259,A -85,B 0,C 180,E1 -14305.249,E2 -14305.249} C_VEL
LIN {X 0,Y 339.188,Z 380.659,A -85,B 0,C 180,E1 -14306.436,E2 -14306.436} C_VEL
LIN {X 0,Y 339.062,Z 382.264,A -85,B 0,C 180,E1 -14308.812,E2 -14308.812} C_VEL
LIN {X 0,Y 339.071,Z 382.496,A -85,B 0,C 180,E1 -14310,E2 -14310} C_VEL
LIN {X 0,Y 339.062,Z 382.306,A -85,B 0,C 180,E1 -14311.188,E2 -14311.188} C_VEL
LIN {X 0,Y 339.185,Z 380.754,A -85,B 0,C 180,E1 -14313.564,E2 -14313.564} C_VEL
LIN {X 0,Y 339.373,Z 379.396,A -85,B 0,C 180,E1 -14314.752,E2 -14314.752} C_VEL
LIN {X 0,Y 339.718,Z 376.067,A -85,B 0,C 180,E1 -14316.776,E2 -14316.776} C_VEL
LIN {X 0,Y 340.198,Z 371.087,A -85,B 0,C 180,E1 -14318.913,E2 -14318.913} C_VEL
LIN {X 0,Y 341.007,Z 364.65,A -85,B 0,C 180,E1 -14320.99,E2 -14320.99} C_VEL
LIN {X 0,Y 341.932,Z 357.575,A -85,B 0,C 180,E1 -14322.765,E2 -14322.765} C_VEL
LIN {X 0,Y 343.187,Z 348.755,A -85,B 0,C 180,E1 -14324.529,E2 -14324.529} C_VEL
LIN {X 0,Y 344.319,Z 340.117,A -85,B 0,C 180,E1 -14325.93,E2 -14325.93} C_VEL
LIN {X 0,Y 345.41,Z 330.063,A -85,B 0,C 180,E1 -14327.266,E2 -14327.266} C_VEL
LIN {X 0,Y 346.472,Z 320.108,A -85,B 0,C 180,E1 -14328.325,E2 -14328.325} C_VEL
LIN {X 0,Y 347.193,Z 310.674,A -85,B 0,C 180,E1 -14329.149,E2 -14329.149} C_VEL
LIN {X 0,Y 345.065,Z 299.037,A -85,B 0,C 180,E1 -14330.117,E2 -14330.117} C_VEL
LIN {X 0,Y 341.989,Z 286.073,A -85,B 0,C 180,E1 -14330.988,E2 -14330.988} C_VEL
LIN {X 0,Y 339.783,Z 278.136,A -85,B 0,C 180,E1 -14331.444,E2 -14331.444} C_VEL
LIN {X 0,Y 339.998,Z 274.435,A -85,B 0,C 180,E1 -14334.562,E2 -14334.562} C_VEL
LIN {X 0,Y 340.208,Z 271.283,A -85,B 0,C 180,E1 -14337.34,E2 -14337.34} C_VEL
LIN {X 0,Y 340.407,Z 267.167,A -85,B 0,C 180,E1 -14341.074,E2 -14341.074} C_VEL
LIN {X 0,Y 340.649,Z 263.684,A -85,B 0,C 180,E1 -14344.386,E2 -14344.386} C_VEL
LIN {X 0,Y 340.636,Z 261.282,A -85,B 0,C 180,E1 -14346.751,E2 -14346.751} C_VEL
LIN {X 0,Y 340.684,Z 261.049,A -85,B 0,C 180,E1 -14348.38,E2 -14348.38} C_VEL
LIN {X 0,Y 340.695,Z 261.045,A -85,B 0,C 180,E1 -14352.044,E2 -14352.044} C_VEL
LIN {X 0,Y 340.653,Z 261.053,A -85,B 0,C 180,E1 -14356.227,E2 -14356.227} C_VEL
LIN {X 0,Y 340.695,Z 261.046,A -85,B 0,C 180,E1 -14358.018,E2 -14358.018} C_VEL
LIN {X 0,Y 340.004,Z 261.131,A -85,B 0,C 180,E1 -14359.005,E2 -14359.005} C_VEL
LIN {X 0,Y 337.162,Z 261.486,A -85,B 0,C 180,E1 -14360.611,E2 -14360.611} C_VEL
LIN {X 0,Y 334.772,Z 261.785,A -85,B 0,C 180,E1 -14361.911,E2 -14361.911} C_VEL
LIN {X 0,Y 333.749,Z 261.909,A -85,B 0,C 180,E1 -14362.917,E2 -14362.917} C_VEL
LIN {X 0,Y 333.666,Z 261.919,A -85,B 0,C 180,E1 -14363.258,E2 -14363.258} C_VEL
LIN {X 0,Y 333.639,Z 261.923,A -85,B 0,C 180,E1 -14366.792,E2 -14366.792} C_VEL
LIN {X 0,Y 333.705,Z 261.918,A -85,B 0,C 180,E1 -14369.71,E2 -14369.71} C_VEL
LIN {X 0,Y 333.746,Z 261.909,A -85,B 0,C 180,E1 -14372.401,E2 -14372.401} C_VEL
LIN {X 0,Y 333.728,Z 261.913,A -85,B 0,C 180,E1 -14375.091,E2 -14375.091} C_VEL
LIN {X 0,Y 333.673,Z 261.92,A -85,B 0,C 180,E1 -14379.019,E2 -14379.019} C_VEL
LIN {X 0,Y 333.743,Z 261.914,A -85,B 0,C 180,E1 -14381.586,E2 -14381.586} C_VEL
LIN {X 0,Y 333.811,Z 261.904,A -85,B 0,C 180,E1 -14385.577,E2 -14385.577} C_VEL
LIN {X 0,Y 333.821,Z 261.904,A -85,B 0,C 180,E1 -14389.078,E2 -14389.078} C_VEL
LIN {X 0,Y 333.974,Z 261.884,A -85,B 0,C 180,E1 -14392.746,E2 -14392.746} C_VEL
LIN {X 0,Y 333.793,Z 261.907,A -85,B 0,C 180,E1 -14395.169,E2 -14395.169} C_VEL
LIN {X 0,Y 334.072,Z 261.869,A -85,B 0,C 180,E1 -14397.589,E2 -14397.589} C_VEL
LIN {X 0,Y 334.086,Z 261.869,A -85,B 0,C 180,E1 -14401.205,E2 -14401.205} C_VEL
LIN {X 0,Y 334.108,Z 261.867,A -85,B 0,C 180,E1 -14402.411,E2 -14402.411} C_VEL
LIN {X 0,Y 334.011,Z 261.877,A -85,B 0,C 180,E1 -14406.039,E2 -14406.039} C_VEL
LIN {X 0,Y 333.821,Z 261.9,A -85,B 0,C 180,E1 -14409.696,E2 -14409.696} C_VEL
LIN {X 0,Y 333.798,Z 261.903,A -85,B 0,C 180,E1 -14413.391,E2 -14413.391} C_VEL
LIN {X 0,Y 333.749,Z 261.909,A -85,B 0,C 180,E1 -14417.146,E2 -14417.146} C_VEL
LIN {X 0,Y 333.737,Z 261.912,A -85,B 0,C 180,E1 -14419.69,E2 -14419.69} C_VEL
LIN {X 0,Y 333.647,Z 261.924,A -85,B 0,C 180,E1 -14423.592,E2 -14423.592} C_VEL
LIN {X 0,Y 333.67,Z 261.922,A -85,B 0,C 180,E1 -14427.605,E2 -14427.605} C_VEL
LIN {X 0,Y 333.66,Z 261.921,A -85,B 0,C 180,E1 -14430.366,E2 -14430.366} C_VEL
LIN {X 0,Y 333.641,Z 261.925,A -85,B 0,C 180,E1 -14433.208,E2 -14433.208} C_VEL
LIN {X 0,Y 333.677,Z 261.92,A -85,B 0,C 180,E1 -14436.139,E2 -14436.139} C_VEL
LIN {X 0,Y 333.621,Z 261.929,A -85,B 0,C 180,E1 -14439.196,E2 -14439.196} C_VEL
LIN {X 0,Y 333.63,Z 261.925,A -85,B 0,C 180,E1 -14442.499,E2 -14442.499} C_VEL
LIN {X 0,Y 333.67,Z 262.047,A -85,B 0,C 180,E1 -14445.736,E2 -14445.736} C_VEL
LIN {X 0,Y 334.447,Z 266.317,A -85,B 0,C 180,E1 -14449.156,E2 -14449.156} C_VEL
LIN {X 0,Y 335.089,Z 270.83,A -85,B 0,C 180,E1 -14452.538,E2 -14452.538} C_VEL
LIN {X 0,Y 335.189,Z 274.143,A -85,B 0,C 180,E1 -14454.858,E2 -14454.858} C_VEL
LIN {X 0,Y 334.559,Z 279.349,A -85,B 0,C 180,E1 -14458.32,E2 -14458.32} C_VEL
LIN {X 0,Y 333.815,Z 285.679,A -85,B 0,C 180,E1 -14462.407,E2 -14462.407} C_VEL
LIN {X 0,Y 333.221,Z 291.961,A -85,B 0,C 180,E1 -14466.376,E2 -14466.376} C_VEL
LIN {X 0,Y 333.021,Z 294.762,A -85,B 0,C 180,E1 -14468.132,E2 -14468.132} C_VEL
LIN {X 0,Y 335.99,Z 308.41,A -85,B 0,C 180,E1 -14468.873,E2 -14468.873} C_VEL
LIN {X 0,Y 338.087,Z 321.199,A -85,B 0,C 180,E1 -14469.773,E2 -14469.773} C_VEL
LIN {X 0,Y 339.263,Z 333.084,A -85,B 0,C 180,E1 -14470.8,E2 -14470.8} C_VEL
LIN {X 0,Y 338.88,Z 339.472,A -85,B 0,C 180,E1 -14471.406,E2 -14471.406} C_VEL
LIN {X 0,Y 337.566,Z 350.082,A -85,B 0,C 180,E1 -14472.585,E2 -14472.585} C_VEL
LIN {X 0,Y 336.167,Z 360.859,A -85,B 0,C 180,E1 -14474.09,E2 -14474.09} C_VEL
LIN {X 0,Y 335.089,Z 370.209,A -85,B 0,C 180,E1 -14475.733,E2 -14475.733} C_VEL
LIN {X 0,Y 333.898,Z 378.481,A -85,B 0,C 180,E1 -14477.541,E2 -14477.541} C_VEL
LIN {X 0,Y 333.111,Z 385.154,A -85,B 0,C 180,E1 -14479.362,E2 -14479.362} C_VEL
LIN {X 0,Y 332.463,Z 391.261,A -85,B 0,C 180,E1 -14481.49,E2 -14481.49} C_VEL
LIN {X 0,Y 332.123,Z 395.231,A -85,B 0,C 180,E1 -14483.316,E2 -14483.316} C_VEL
LIN {X 0,Y 331.986,Z 398.167,A -85,B 0,C 180,E1 -14485.142,E2 -14485.142} C_VEL
LIN {X 0,Y 331.996,Z 399.564,A -85,B 0,C 180,E1 -14486.359,E2 -14486.359} C_VEL
LIN {X 0,Y 331.923,Z 401.168,A -85,B 0,C 180,E1 -14488.787,E2 -14488.787} C_VEL
LIN {X 0,Y 331.97,Z 401.383,A -85,B 0,C 180,E1 -14490,E2 -14490} C_VEL
LIN {X 0,Y 331.923,Z 401.163,A -85,B 0,C 180,E1 -14491.213,E2 -14491.213} C_VEL
LIN {X 0,Y 331.991,Z 399.553,A -85,B 0,C 180,E1 -14493.641,E2 -14493.641} C_VEL
LIN {X 0,Y 332.006,Z 396.784,A -85,B 0,C 180,E1 -14495.782,E2 -14495.782} C_VEL
LIN {X 0,Y 332.333,Z 392.658,A -85,B 0,C 180,E1 -14497.901,E2 -14497.901} C_VEL
LIN {X 0,Y 332.79,Z 387.926,A -85,B 0,C 180,E1 -14499.727,E2 -14499.727} C_VEL
LIN {X 0,Y 333.435,Z 381.941,A -85,B 0,C 180,E1 -14501.551,E2 -14501.551} C_VEL
LIN {X 0,Y 334.479,Z 374.495,A -85,B 0,C 180,E1 -14503.363,E2 -14503.363} C_VEL
LIN {X 0,Y 335.46,Z 366.905,A -85,B 0,C 180,E1 -14504.871,E2 -14504.871} C_VEL
LIN {X 0,Y 336.694,Z 356.989,A -85,B 0,C 180,E1 -14506.476,E2 -14506.476} C_VEL
LIN {X 0,Y 337.996,Z 346.212,A -85,B 0,C 180,E1 -14507.86,E2 -14507.86} C_VEL
LIN {X 0,Y 339.285,Z 334.597,A -85,B 0,C 180,E1 -14509.041,E2 -14509.041} C_VEL
LIN {X 0,Y 338.41,Z 324.119,A -85,B 0,C 180,E1 -14509.981,E2 -14509.981} C_VEL
LIN {X 0,Y 336.56,Z 311.906,A -85,B 0,C 180,E1 -14510.888,E2 -14510.888} C_VEL
LIN {X 0,Y 333.95,Z 299.16,A -85,B 0,C 180,E1 -14511.635,E2 -14511.635} C_VEL
LIN {X 0,Y 332.999,Z 294.726,A -85,B 0,C 180,E1 -14511.873,E2 -14511.873} C_VEL
LIN {X 0,Y 333.507,Z 288.803,A -85,B 0,C 180,E1 -14515.594,E2 -14515.594} C_VEL
LIN {X 0,Y 334.164,Z 282.474,A -85,B 0,C 180,E1 -14519.62,E2 -14519.62} C_VEL
LIN {X 0,Y 334.787,Z 277.174,A -85,B 0,C 180,E1 -14523.08,E2 -14523.08} C_VEL
LIN {X 0,Y 335.175,Z 272.904,A -85,B 0,C 180,E1 -14525.952,E2 -14525.952} C_VEL
LIN {X 0,Y 334.8,Z 268.623,A -85,B 0,C 180,E1 -14529.041,E2 -14529.041} C_VEL
LIN {X 0,Y 334.078,Z 264.063,A -85,B 0,C 180,E1 -14532.583,E2 -14532.583} C_VEL
LIN {X 0,Y 333.647,Z 261.928,A -85,B 0,C 180,E1 -14534.462,E2 -14534.462} C_VEL
LIN {X 0,Y 333.638,Z 261.923,A -85,B 0,C 180,E1 -14537.618,E2 -14537.618} C_VEL
LIN {X 0,Y 333.634,Z 261.925,A -85,B 0,C 180,E1 -14541.206,E2 -14541.206} C_VEL
LIN {X 0,Y 333.676,Z 261.919,A -85,B 0,C 180,E1 -14543.861,E2 -14543.861} C_VEL
LIN {X 0,Y 333.647,Z 261.923,A -85,B 0,C 180,E1 -14547.412,E2 -14547.412} C_VEL
LIN {X 0,Y 333.655,Z 261.922,A -85,B 0,C 180,E1 -14551.023,E2 -14551.023} C_VEL
LIN {X 0,Y 333.667,Z 261.92,A -85,B 0,C 180,E1 -14555.086,E2 -14555.086} C_VEL
LIN {X 0,Y 333.669,Z 261.919,A -85,B 0,C 180,E1 -14559.018,E2 -14559.018} C_VEL
LIN {X 0,Y 333.796,Z 261.906,A -85,B 0,C 180,E1 -14561.59,E2 -14561.59} C_VEL
LIN {X 0,Y 333.81,Z 261.905,A -85,B 0,C 180,E1 -14565.577,E2 -14565.577} C_VEL
LIN {X 0,Y 333.818,Z 261.901,A -85,B 0,C 180,E1 -14569.078,E2 -14569.078} C_VEL
LIN {X 0,Y 333.994,Z 261.879,A -85,B 0,C 180,E1 -14572.747,E2 -14572.747} C_VEL
LIN {X 0,Y 333.808,Z 261.905,A -85,B 0,C 180,E1 -14575.169,E2 -14575.169} C_VEL
LIN {X 0,Y 334.106,Z 261.867,A -85,B 0,C 180,E1 -14577.589,E2 -14577.589} C_VEL
LIN {X 0,Y 334.207,Z 261.852,A -85,B 0,C 180,E1 -14580,E2 -14580} C_VEL
LIN {X 0,Y 334.071,Z 261.869,A -85,B 0,C 180,E1 -14582.411,E2 -14582.411} C_VEL
LIN {X 0,Y 333.978,Z 261.879,A -85,B 0,C 180,E1 -14586.624,E2 -14586.624} C_VEL
LIN {X 0,Y 333.822,Z 261.9,A -85,B 0,C 180,E1 -14589.696,E2 -14589.696} C_VEL
LIN {X 0,Y 333.798,Z 261.904,A -85,B 0,C 180,E1 -14593.391,E2 -14593.391} C_VEL
LIN {X 0,Y 333.72,Z 261.914,A -85,B 0,C 180,E1 -14597.148,E2 -14597.148} C_VEL
LIN {X 0,Y 333.687,Z 261.917,A -85,B 0,C 180,E1 -14599.694,E2 -14599.694} C_VEL
LIN {X 0,Y 333.67,Z 261.919,A -85,B 0,C 180,E1 -14603.59,E2 -14603.59} C_VEL
LIN {X 0,Y 333.737,Z 261.915,A -85,B 0,C 180,E1 -14606.246,E2 -14606.246} C_VEL
LIN {X 0,Y 333.712,Z 261.914,A -85,B 0,C 180,E1 -14608.972,E2 -14608.972} C_VEL
LIN {X 0,Y 333.644,Z 261.924,A -85,B 0,C 180,E1 -14612.587,E2 -14612.587} C_VEL
LIN {X 0,Y 333.675,Z 261.923,A -85,B 0,C 180,E1 -14616.139,E2 -14616.139} C_VEL
LIN {X 0,Y 333.647,Z 261.922,A -85,B 0,C 180,E1 -14619.193,E2 -14619.193} C_VEL
LIN {X 0,Y 333.632,Z 261.924,A -85,B 0,C 180,E1 -14622.5,E2 -14622.5} C_VEL
LIN {X 0,Y 333.595,Z 261.931,A -85,B 0,C 180,E1 -14625.955,E2 -14625.955} C_VEL
LIN {X 0,Y 333.602,Z 261.932,A -85,B 0,C 180,E1 -14629.325,E2 -14629.325} C_VEL
LIN {X 0,Y 333.624,Z 261.929,A -85,B 0,C 180,E1 -14632.345,E2 -14632.345} C_VEL
LIN {X 0,Y 333.622,Z 262.134,A -85,B 0,C 180,E1 -14633.178,E2 -14633.178} C_VEL
LIN {X 0,Y 333.653,Z 264.269,A -85,B 0,C 180,E1 -14635.339,E2 -14635.339} C_VEL
LIN {X 0,Y 333.436,Z 267.217,A -85,B 0,C 180,E1 -14638.201,E2 -14638.201} C_VEL
LIN {X 0,Y 333.263,Z 270.192,A -85,B 0,C 180,E1 -14640.985,E2 -14640.985} C_VEL
LIN {X 0,Y 333.063,Z 273.168,A -85,B 0,C 180,E1 -14643.697,E2 -14643.697} C_VEL
LIN {X 0,Y 332.751,Z 277.704,A -85,B 0,C 180,E1 -14647.655,E2 -14647.655} C_VEL
LIN {X 0,Y 332.731,Z 278.347,A -85,B 0,C 180,E1 -14648.206,E2 -14648.206} C_VEL
LIN {X 0,Y 336.395,Z 291.712,A -85,B 0,C 180,E1 -14649.014,E2 -14649.014} C_VEL
LIN {X 0,Y 339.03,Z 303.907,A -85,B 0,C 180,E1 -14649.937,E2 -14649.937} C_VEL
LIN {X 0,Y 340.422,Z 312.556,A -85,B 0,C 180,E1 -14650.712,E2 -14650.712} C_VEL
LIN {X 0,Y 339.319,Z 323.65,A -85,B 0,C 180,E1 -14651.744,E2 -14651.744} C_VEL
LIN {X 0,Y 338.266,Z 333.441,A -85,B 0,C 180,E1 -14652.887,E2 -14652.887} C_VEL
LIN {X 0,Y 337.076,Z 343.118,A -85,B 0,C 180,E1 -14654.273,E2 -14654.273} C_VEL
LIN {X 0,Y 335.891,Z 351.61,A -85,B 0,C 180,E1 -14655.768,E2 -14655.768} C_VEL
LIN {X 0,Y 334.767,Z 359.86,A -85,B 0,C 180,E1 -14657.574,E2 -14657.574} C_VEL
LIN {X 0,Y 333.828,Z 366.506,A -85,B 0,C 180,E1 -14659.385,E2 -14659.385} C_VEL
LIN {X 0,Y 332.99,Z 372.594,A -85,B 0,C 180,E1 -14661.504,E2 -14661.504} C_VEL
LIN {X 0,Y 332.557,Z 376.583,A -85,B 0,C 180,E1 -14663.347,E2 -14663.347} C_VEL
LIN {X 0,Y 332.303,Z 379.46,A -85,B 0,C 180,E1 -14665.147,E2 -14665.147} C_VEL
LIN {X 0,Y 332.119,Z 380.859,A -85,B 0,C 180,E1 -14666.36,E2 -14666.36} C_VEL
LIN {X 0,Y 331.967,Z 382.464,A -85,B 0,C 180,E1 -14668.787,E2 -14668.787} C_VEL
LIN {X 0,Y 331.975,Z 382.695,A -85,B 0,C 180,E1 -14670,E2 -14670} C_VEL
LIN {X 0,Y 331.967,Z 382.505,A -85,B 0,C 180,E1 -14671.213,E2 -14671.213} C_VEL
LIN {X 0,Y 332.117,Z 380.953,A -85,B 0,C 180,E1 -14673.64,E2 -14673.64} C_VEL
LIN {X 0,Y 332.295,Z 379.595,A -85,B 0,C 180,E1 -14674.853,E2 -14674.853} C_VEL
LIN {X 0,Y 332.609,Z 376.632,A -85,B 0,C 180,E1 -14676.729,E2 -14676.729} C_VEL
LIN {X 0,Y 332.995,Z 372.843,A -85,B 0,C 180,E1 -14678.496,E2 -14678.496} C_VEL
LIN {X 0,Y 333.636,Z 367.827,A -85,B 0,C 180,E1 -14680.315,E2 -14680.315} C_VEL
LIN {X 0,Y 334.517,Z 361.51,A -85,B 0,C 180,E1 -14682.128,E2 -14682.128} C_VEL
LIN {X 0,Y 335.629,Z 353.602,A -85,B 0,C 180,E1 -14683.934,E2 -14683.934} C_VEL
LIN {X 0,Y 336.789,Z 345.538,A -85,B 0,C 180,E1 -14685.43,E2 -14685.43} C_VEL
LIN {X 0,Y 338.024,Z 335.311,A -85,B 0,C 180,E1 -14686.979,E2 -14686.979} C_VEL
LIN {X 0,Y 339.207,Z 324.627,A -85,B 0,C 180,E1 -14688.263,E2 -14688.263} C_VEL
LIN {X 0,Y 340.375,Z 313.766,A -85,B 0,C 180,E1 -14689.291,E2 -14689.291} C_VEL
LIN {X 0,Y 340.167,Z 310.138,A -85,B 0,C 180,E1 -14689.621,E2 -14689.621} C_VEL
LIN {X 0,Y 337.913,Z 298.264,A -85,B 0,C 180,E1 -14690.622,E2 -14690.622} C_VEL
LIN {X 0,Y 334.811,Z 285.706,A -85,B 0,C 180,E1 -14691.485,E2 -14691.485} C_VEL
LIN {X 0,Y 332.743,Z 278.312,A -85,B 0,C 180,E1 -14691.934,E2 -14691.934} C_VEL
LIN {X 0,Y 332.951,Z 274.791,A -85,B 0,C 180,E1 -14694.972,E2 -14694.972} C_VEL
LIN {X 0,Y 333.175,Z 271.814,A -85,B 0,C 180,E1 -14697.65,E2 -14697.65} C_VEL
LIN {X 0,Y 333.409,Z 267.341,A -85,B 0,C 180,E1 -14701.802,E2 -14701.802} C_VEL
LIN {X 0,Y 333.617,Z 264.297,A -85,B 0,C 180,E1 -14704.757,E2 -14704.757} C_VEL
LIN {X 0,Y 333.605,Z 262.26,A -85,B 0,C 180,E1 -14706.818,E2 -14706.818} C_VEL
LIN {X 0,Y 333.611,Z 261.929,A -85,B 0,C 180,E1 -14708.788,E2 -14708.788} C_VEL
LIN {X 0,Y 333.63,Z 261.928,A -85,B 0,C 180,E1 -14712.499,E2 -14712.499} C_VEL
LIN {X 0,Y 333.597,Z 261.929,A -85,B 0,C 180,E1 -14715.955,E2 -14715.955} C_VEL
LIN {X 0,Y 333.648,Z 261.922,A -85,B 0,C 180,E1 -14719.316,E2 -14719.316} C_VEL
LIN {X 0,Y 333.666,Z 261.919,A -85,B 0,C 180,E1 -14723.258,E2 -14723.258} C_VEL
LIN {X 0,Y 332.989,Z 262.008,A -85,B 0,C 180,E1 -14724.265,E2 -14724.265} C_VEL
LIN {X 0,Y 330.104,Z 262.368,A -85,B 0,C 180,E1 -14725.904,E2 -14725.904} C_VEL
LIN {X 0,Y 327.675,Z 262.666,A -85,B 0,C 180,E1 -14727.231,E2 -14727.231} C_VEL
LIN {X 0,Y 326.654,Z 262.795,A -85,B 0,C 180,E1 -14728.259,E2 -14728.259} C_VEL
LIN {X 0,Y 326.582,Z 262.799,A -85,B 0,C 180,E1 -14728.607,E2 -14728.607} C_VEL
LIN {X 0,Y 326.663,Z 262.795,A -85,B 0,C 180,E1 -14731.897,E2 -14731.897} C_VEL
LIN {X 0,Y 326.69,Z 262.788,A -85,B 0,C 180,E1 -14734.627,E2 -14734.627} C_VEL
LIN {X 0,Y 326.62,Z 262.797,A -85,B 0,C 180,E1 -14738.543,E2 -14738.543} C_VEL
LIN {X 0,Y 326.709,Z 262.789,A -85,B 0,C 180,E1 -14741.175,E2 -14741.175} C_VEL
LIN {X 0,Y 326.766,Z 262.783,A -85,B 0,C 180,E1 -14745.433,E2 -14745.433} C_VEL
LIN {X 0,Y 326.762,Z 262.781,A -85,B 0,C 180,E1 -14748.839,E2 -14748.839} C_VEL
LIN {X 0,Y 326.928,Z 262.76,A -85,B 0,C 180,E1 -14752.589,E2 -14752.589} C_VEL
LIN {X 0,Y 326.761,Z 262.784,A -85,B 0,C 180,E1 -14755.065,E2 -14755.065} C_VEL
LIN {X 0,Y 327.016,Z 262.748,A -85,B 0,C 180,E1 -14757.536,E2 -14757.536} C_VEL
LIN {X 0,Y 327.054,Z 262.744,A -85,B 0,C 180,E1 -14761.231,E2 -14761.231} C_VEL
LIN {X 0,Y 327.048,Z 262.747,A -85,B 0,C 180,E1 -14762.463,E2 -14762.463} C_VEL
LIN {X 0,Y 326.985,Z 262.754,A -85,B 0,C 180,E1 -14766.169,E2 -14766.169} C_VEL
LIN {X 0,Y 326.784,Z 262.778,A -85,B 0,C 180,E1 -14769.907,E2 -14769.907} C_VEL
LIN {X 0,Y 326.761,Z 262.78,A -85,B 0,C 180,E1 -14773.685,E2 -14773.685} C_VEL
LIN {X 0,Y 326.702,Z 262.787,A -85,B 0,C 180,E1 -14777.528,E2 -14777.528} C_VEL
LIN {X 0,Y 326.663,Z 262.797,A -85,B 0,C 180,E1 -14780.135,E2 -14780.135} C_VEL
LIN {X 0,Y 326.614,Z 262.802,A -85,B 0,C 180,E1 -14784.132,E2 -14784.132} C_VEL
LIN {X 0,Y 326.601,Z 262.802,A -85,B 0,C 180,E1 -14788.256,E2 -14788.256} C_VEL
LIN {X 0,Y 326.576,Z 262.804,A -85,B 0,C 180,E1 -14791.097,E2 -14791.097} C_VEL
LIN {X 0,Y 326.61,Z 262.801,A -85,B 0,C 180,E1 -14794.019,E2 -14794.019} C_VEL
LIN {X 0,Y 326.625,Z 262.801,A -85,B 0,C 180,E1 -14797.237,E2 -14797.237} C_VEL
LIN {X 0,Y 326.546,Z 262.811,A -85,B 0,C 180,E1 -14801.124,E2 -14801.124} C_VEL
LIN {X 0,Y 326.57,Z 262.808,A -85,B 0,C 180,E1 -14804.946,E2 -14804.946} C_VEL
LIN {X 0,Y 326.572,Z 262.807,A -85,B 0,C 180,E1 -14805.25,E2 -14805.25} C_VEL
LIN {X 0,Y 327.361,Z 266.97,A -85,B 0,C 180,E1 -14808.712,E2 -14808.712} C_VEL
LIN {X 0,Y 327.97,Z 270.681,A -85,B 0,C 180,E1 -14811.579,E2 -14811.579} C_VEL
LIN {X 0,Y 328.17,Z 274.929,A -85,B 0,C 180,E1 -14814.674,E2 -14814.674} C_VEL
LIN {X 0,Y 327.523,Z 280.233,A -85,B 0,C 180,E1 -14818.283,E2 -14818.283} C_VEL
LIN {X 0,Y 326.831,Z 285.604,A -85,B 0,C 180,E1 -14821.841,E2 -14821.841} C_VEL
LIN {X 0,Y 326.21,Z 291.758,A -85,B 0,C 180,E1 -14825.836,E2 -14825.836} C_VEL
LIN {X 0,Y 325.995,Z 294.653,A -85,B 0,C 180,E1 -14827.644,E2 -14827.644} C_VEL
LIN {X 0,Y 328.901,Z 307.643,A -85,B 0,C 180,E1 -14828.364,E2 -14828.364} C_VEL
LIN {X 0,Y 330.969,Z 319.558,A -85,B 0,C 180,E1 -14829.215,E2 -14829.215} C_VEL
LIN {X 0,Y 332.229,Z 331.106,A -85,B 0,C 180,E1 -14830.216,E2 -14830.216} C_VEL
LIN {X 0,Y 332.479,Z 336.16,A -85,B 0,C 180,E1 -14830.714,E2 -14830.714} C_VEL
LIN {X 0,Y 331.098,Z 347.451,A -85,B 0,C 180,E1 -14831.914,E2 -14831.914} C_VEL
LIN {X 0,Y 329.754,Z 357.627,A -85,B 0,C 180,E1 -14833.278,E2 -14833.278} C_VEL
LIN {X 0,Y 328.508,Z 367.046,A -85,B 0,C 180,E1 -14834.856,E2 -14834.856} C_VEL
LIN {X 0,Y 327.349,Z 375.727,A -85,B 0,C 180,E1 -14836.656,E2 -14836.656} C_VEL
LIN {X 0,Y 326.336,Z 382.917,A -85,B 0,C 180,E1 -14838.509,E2 -14838.509} C_VEL
LIN {X 0,Y 325.578,Z 389.47,A -85,B 0,C 180,E1 -14840.683,E2 -14840.683} C_VEL
LIN {X 0,Y 325.152,Z 393.807,A -85,B 0,C 180,E1 -14842.548,E2 -14842.548} C_VEL
LIN {X 0,Y 324.925,Z 396.835,A -85,B 0,C 180,E1 -14844.249,E2 -14844.249} C_VEL
LIN {X 0,Y 324.9,Z 399.365,A -85,B 0,C 180,E1 -14846.279,E2 -14846.279} C_VEL
LIN {X 0,Y 324.831,Z 400.969,A -85,B 0,C 180,E1 -14848.76,E2 -14848.76} C_VEL
LIN {X 0,Y 324.874,Z 401.184,A -85,B 0,C 180,E1 -14850,E2 -14850} C_VEL
LIN {X 0,Y 324.831,Z 400.963,A -85,B 0,C 180,E1 -14851.24,E2 -14851.24} C_VEL
LIN {X 0,Y 324.894,Z 399.353,A -85,B 0,C 180,E1 -14853.721,E2 -14853.721} C_VEL
LIN {X 0,Y 324.91,Z 396.852,A -85,B 0,C 180,E1 -14855.725,E2 -14855.725} C_VEL
LIN {X 0,Y 325.152,Z 393.773,A -85,B 0,C 180,E1 -14857.451,E2 -14857.451} C_VEL
LIN {X 0,Y 325.578,Z 389.424,A -85,B 0,C 180,E1 -14859.317,E2 -14859.317} C_VEL
LIN {X 0,Y 326.216,Z 383.886,A -85,B 0,C 180,E1 -14861.18,E2 -14861.18} C_VEL
LIN {X 0,Y 327.167,Z 376.979,A -85,B 0,C 180,E1 -14863.035,E2 -14863.035} C_VEL
LIN {X 0,Y 328.165,Z 369.927,A -85,B 0,C 180,E1 -14864.574,E2 -14864.574} C_VEL
LIN {X 0,Y 329.337,Z 360.857,A -85,B 0,C 180,E1 -14866.199,E2 -14866.199} C_VEL
LIN {X 0,Y 330.629,Z 350.927,A -85,B 0,C 180,E1 -14867.632,E2 -14867.632} C_VEL
LIN {X 0,Y 332.12,Z 339.112,A -85,B 0,C 180,E1 -14868.987,E2 -14868.987} C_VEL
LIN {X 0,Y 332.438,Z 334.388,A -85,B 0,C 180,E1 -14869.449,E2 -14869.449} C_VEL
LIN {X 0,Y 331.276,Z 322,A -85,B 0,C 180,E1 -14870.57,E2 -14870.57} C_VEL
LIN {X 0,Y 329.078,Z 308.659,A -85,B 0,C 180,E1 -14871.548,E2 -14871.548} C_VEL
LIN {X 0,Y 326.199,Z 295.993,A -85,B 0,C 180,E1 -14872.281,E2 -14872.281} C_VEL
LIN {X 0,Y 325.992,Z 294.551,A -85,B 0,C 180,E1 -14872.348,E2 -14872.348} C_VEL
LIN {X 0,Y 326.522,Z 288.609,A -85,B 0,C 180,E1 -14876.183,E2 -14876.183} C_VEL
LIN {X 0,Y 327.103,Z 283.339,A -85,B 0,C 180,E1 -14879.615,E2 -14879.615} C_VEL
LIN {X 0,Y 327.791,Z 277.906,A -85,B 0,C 180,E1 -14883.261,E2 -14883.261} C_VEL
LIN {X 0,Y 328.151,Z 274.603,A -85,B 0,C 180,E1 -14885.526,E2 -14885.526} C_VEL
LIN {X 0,Y 327.928,Z 270.617,A -85,B 0,C 180,E1 -14888.427,E2 -14888.427} C_VEL
LIN {X 0,Y 327.258,Z 266.376,A -85,B 0,C 180,E1 -14891.739,E2 -14891.739} C_VEL
LIN {X 0,Y 326.567,Z 262.809,A -85,B 0,C 180,E1 -14894.75,E2 -14894.75} C_VEL
LIN {X 0,Y 326.563,Z 262.805,A -85,B 0,C 180,E1 -14898.152,E2 -14898.152} C_VEL
LIN {X 0,Y 326.582,Z 262.803,A -85,B 0,C 180,E1 -14901.386,E2 -14901.386} C_VEL
LIN {X 0,Y 326.62,Z 262.8,A -85,B 0,C 180,E1 -14904.851,E2 -14904.851} C_VEL
LIN {X 0,Y 326.611,Z 262.8,A -85,B 0,C 180,E1 -14907.456,E2 -14907.456} C_VEL
LIN {X 0,Y 326.618,Z 262.803,A -85,B 0,C 180,E1 -14910.337,E2 -14910.337} C_VEL
LIN {X 0,Y 326.603,Z 262.802,A -85,B 0,C 180,E1 -14914.509,E2 -14914.509} C_VEL
LIN {X 0,Y 326.617,Z 262.799,A -85,B 0,C 180,E1 -14918.543,E2 -14918.543} C_VEL
LIN {X 0,Y 326.746,Z 262.782,A -85,B 0,C 180,E1 -14921.178,E2 -14921.178} C_VEL
LIN {X 0,Y 326.764,Z 262.782,A -85,B 0,C 180,E1 -14925.433,E2 -14925.433} C_VEL
LIN {X 0,Y 326.759,Z 262.78,A -85,B 0,C 180,E1 -14928.839,E2 -14928.839} C_VEL
LIN {X 0,Y 326.943,Z 262.756,A -85,B 0,C 180,E1 -14932.59,E2 -14932.59} C_VEL
LIN {X 0,Y 326.984,Z 262.754,A -85,B 0,C 180,E1 -14933.831,E2 -14933.831} C_VEL
LIN {X 0,Y 327.047,Z 262.747,A -85,B 0,C 180,E1 -14937.537,E2 -14937.537} C_VEL
LIN {X 0,Y 327.16,Z 262.73,A -85,B 0,C 180,E1 -14940,E2 -14940} C_VEL
LIN {X 0,Y 327.015,Z 262.748,A -85,B 0,C 180,E1 -14942.464,E2 -14942.464} C_VEL
LIN {X 0,Y 326.935,Z 262.756,A -85,B 0,C 180,E1 -14946.617,E2 -14946.617} C_VEL
LIN {X 0,Y 326.785,Z 262.776,A -85,B 0,C 180,E1 -14949.907,E2 -14949.907} C_VEL
LIN {X 0,Y 326.761,Z 262.78,A -85,B 0,C 180,E1 -14953.685,E2 -14953.685} C_VEL
LIN {X 0,Y 326.665,Z 262.791,A -85,B 0,C 180,E1 -14957.53,E2 -14957.53} C_VEL
LIN {X 0,Y 326.632,Z 262.798,A -85,B 0,C 180,E1 -14960.137,E2 -14960.137} C_VEL
LIN {X 0,Y 326.65,Z 262.796,A -85,B 0,C 180,E1 -14964.129,E2 -14964.129} C_VEL
LIN {X 0,Y 326.686,Z 262.79,A -85,B 0,C 180,E1 -14966.858,E2 -14966.858} C_VEL
LIN {X 0,Y 326.64,Z 262.796,A -85,B 0,C 180,E1 -14970.611,E2 -14970.611} C_VEL
LIN {X 0,Y 326.607,Z 262.804,A -85,B 0,C 180,E1 -14974.02,E2 -14974.02} C_VEL
LIN {X 0,Y 326.627,Z 262.797,A -85,B 0,C 180,E1 -14977.238,E2 -14977.238} C_VEL
LIN {X 0,Y 326.577,Z 262.803,A -85,B 0,C 180,E1 -14981.131,E2 -14981.131} C_VEL
LIN {X 0,Y 326.527,Z 262.809,A -85,B 0,C 180,E1 -14984.743,E2 -14984.743} C_VEL
LIN {X 0,Y 326.561,Z 262.807,A -85,B 0,C 180,E1 -14988.152,E2 -14988.152} C_VEL
LIN {X 0,Y 326.561,Z 262.81,A -85,B 0,C 180,E1 -14991.383,E2 -14991.383} C_VEL
LIN {X 0,Y 326.594,Z 262.956,A -85,B 0,C 180,E1 -14992.948,E2 -14992.948} C_VEL
LIN {X 0,Y 326.552,Z 265.918,A -85,B 0,C 180,E1 -14995.974,E2 -14995.974} C_VEL
LIN {X 0,Y 326.32,Z 269.515,A -85,B 0,C 180,E1 -14999.484,E2 -14999.484} C_VEL
LIN {X 0,Y 326.045,Z 273.355,A -85,B 0,C 180,E1 -15003.085,E2 -15003.085} C_VEL
LIN {X 0,Y 325.822,Z 276.381,A -85,B 0,C 180,E1 -15005.806,E2 -15005.806} C_VEL
LIN {X 0,Y 325.701,Z 278.638,A -85,B 0,C 180,E1 -15007.716,E2 -15007.716} C_VEL
LIN {X 0,Y 329.434,Z 291.91,A -85,B 0,C 180,E1 -15008.548,E2 -15008.548} C_VEL
LIN {X 0,Y 332.215,Z 304.699,A -85,B 0,C 180,E1 -15009.549,E2 -15009.549} C_VEL
LIN {X 0,Y 333.63,Z 312.765,A -85,B 0,C 180,E1 -15010.303,E2 -15010.303} C_VEL
LIN {X 0,Y 332.578,Z 323.855,A -85,B 0,C 180,E1 -15011.36,E2 -15011.36} C_VEL
LIN {X 0,Y 331.317,Z 335.157,A -85,B 0,C 180,E1 -15012.724,E2 -15012.724} C_VEL
LIN {X 0,Y 329.986,Z 345.129,A -85,B 0,C 180,E1 -15014.244,E2 -15014.244} C_VEL
LIN {X 0,Y 328.606,Z 354.77,A -85,B 0,C 180,E1 -15016.078,E2 -15016.078} C_VEL
LIN {X 0,Y 327.432,Z 362.459,A -85,B 0,C 180,E1 -15017.92,E2 -15017.92} C_VEL
LIN {X 0,Y 326.409,Z 369.514,A -85,B 0,C 180,E1 -15020.081,E2 -15020.081} C_VEL
LIN {X 0,Y 325.774,Z 374.211,A -85,B 0,C 180,E1 -15021.939,E2 -15021.939} C_VEL
LIN {X 0,Y 325.394,Z 377.805,A -85,B 0,C 180,E1 -15023.801,E2 -15023.801} C_VEL
LIN {X 0,Y 325.229,Z 379.66,A -85,B 0,C 180,E1 -15025.041,E2 -15025.041} C_VEL
LIN {X 0,Y 325.053,Z 381.058,A -85,B 0,C 180,E1 -15026.281,E2 -15026.281} C_VEL
LIN {X 0,Y 324.875,Z 382.664,A -85,B 0,C 180,E1 -15028.761,E2 -15028.761} C_VEL
LIN {X 0,Y 324.88,Z 382.895,A -85,B 0,C 180,E1 -15030,E2 -15030} C_VEL
LIN {X 0,Y 324.875,Z 382.705,A -85,B 0,C 180,E1 -15031.24,E2 -15031.24} C_VEL
LIN {X 0,Y 325.05,Z 381.151,A -85,B 0,C 180,E1 -15033.719,E2 -15033.719} C_VEL
LIN {X 0,Y 325.222,Z 379.794,A -85,B 0,C 180,E1 -15034.959,E2 -15034.959} C_VEL
LIN {X 0,Y 325.509,Z 377.14,A -85,B 0,C 180,E1 -15036.695,E2 -15036.695} C_VEL
LIN {X 0,Y 325.952,Z 373.042,A -85,B 0,C 180,E1 -15038.681,E2 -15038.681} C_VEL
LIN {X 0,Y 326.651,Z 368.025,A -85,B 0,C 180,E1 -15040.538,E2 -15040.538} C_VEL
LIN {X 0,Y 327.582,Z 361.707,A -85,B 0,C 180,E1 -15042.389,E2 -15042.389} C_VEL
LIN {X 0,Y 328.726,Z 353.8,A -85,B 0,C 180,E1 -15044.233,E2 -15044.233} C_VEL
LIN {X 0,Y 330.231,Z 343.958,A -85,B 0,C 180,E1 -15046.062,E2 -15046.062} C_VEL
LIN {X 0,Y 331.479,Z 333.631,A -85,B 0,C 180,E1 -15047.586,E2 -15047.586} C_VEL
LIN {X 0,Y 332.673,Z 323.399,A -85,B 0,C 180,E1 -15048.794,E2 -15048.794} C_VEL
LIN {X 0,Y 333.657,Z 313.961,A -85,B 0,C 180,E1 -15049.695,E2 -15049.695} C_VEL
LIN {X 0,Y 332.048,Z 303.689,A -85,B 0,C 180,E1 -15050.645,E2 -15050.645} C_VEL
LIN {X 0,Y 329.127,Z 290.607,A -85,B 0,C 180,E1 -15051.655,E2 -15051.655} C_VEL
LIN {X 0,Y 325.702,Z 278.559,A -85,B 0,C 180,E1 -15052.403,E2 -15052.403} C_VEL
LIN {X 0,Y 325.936,Z 274.983,A -85,B 0,C 180,E1 -15055.547,E2 -15055.547} C_VEL
LIN {X 0,Y 326.149,Z 272.003,A -85,B 0,C 180,E1 -15058.299,E2 -15058.299} C_VEL
LIN {X 0,Y 326.467,Z 267.512,A -85,B 0,C 180,E1 -15062.56,E2 -15062.56} C_VEL
LIN {X 0,Y 326.579,Z 264.556,A -85,B 0,C 180,E1 -15065.524,E2 -15065.524} C_VEL
LIN {X 0,Y 326.55,Z 262.923,A -85,B 0,C 180,E1 -15067.22,E2 -15067.22} C_VEL
LIN {X 0,Y 326.552,Z 262.807,A -85,B 0,C 180,E1 -15070.215,E2 -15070.215} C_VEL
LIN {X 0,Y 326.562,Z 262.803,A -85,B 0,C 180,E1 -15073.526,E2 -15073.526} C_VEL
LIN {X 0,Y 326.577,Z 262.803,A -85,B 0,C 180,E1 -15077.028,E2 -15077.028} C_VEL
LIN {X 0,Y 326.613,Z 262.799,A -85,B 0,C 180,E1 -15080.773,E2 -15080.773} C_VEL
LIN {X 0,Y 326.615,Z 262.8,A -85,B 0,C 180,E1 -15084.48,E2 -15084.48} C_VEL
LIN {X 0,Y 326.61,Z 262.8,A -85,B 0,C 180,E1 -15087.456,E2 -15087.456} C_VEL
LIN {X 0,Y 326.582,Z 262.799,A -85,B 0,C 180,E1 -15088.607,E2 -15088.607} C_VEL
LIN {X 0,Y 325.953,Z 262.883,A -85,B 0,C 180,E1 -15089.637,E2 -15089.637} C_VEL
LIN {X 0,Y 323.144,Z 263.239,A -85,B 0,C 180,E1 -15091.314,E2 -15091.314} C_VEL
LIN {X 0,Y 320.746,Z 263.538,A -85,B 0,C 180,E1 -15092.673,E2 -15092.673} C_VEL
LIN {X 0,Y 319.718,Z 263.662,A -85,B 0,C 180,E1 -15093.724,E2 -15093.724} C_VEL
LIN {X 0,Y 319.635,Z 263.67,A -85,B 0,C 180,E1 -15094.08,E2 -15094.08} C_VEL
LIN {X 0,Y 319.57,Z 263.677,A -85,B 0,C 180,E1 -15098.046,E2 -15098.046} C_VEL
LIN {X 0,Y 319.627,Z 263.669,A -85,B 0,C 180,E1 -15102.071,E2 -15102.071} C_VEL
LIN {X 0,Y 319.735,Z 263.655,A -85,B 0,C 180,E1 -15106.008,E2 -15106.008} C_VEL
LIN {X 0,Y 319.738,Z 263.655,A -85,B 0,C 180,E1 -15109.872,E2 -15109.872} C_VEL
LIN {X 0,Y 319.913,Z 263.633,A -85,B 0,C 180,E1 -15113.694,E2 -15113.694} C_VEL
LIN {X 0,Y 319.962,Z 263.627,A -85,B 0,C 180,E1 -15117.482,E2 -15117.482} C_VEL
LIN {X 0,Y 320.022,Z 263.62,A -85,B 0,C 180,E1 -15121.258,E2 -15121.258} C_VEL
LIN {X 0,Y 319.743,Z 263.654,A -85,B 0,C 180,E1 -15123.781,E2 -15123.781} C_VEL
LIN {X 0,Y 319.938,Z 263.632,A -85,B 0,C 180,E1 -15126.306,E2 -15126.306} C_VEL
LIN {X 0,Y 319.736,Z 263.657,A -85,B 0,C 180,E1 -15130.128,E2 -15130.128} C_VEL
LIN {X 0,Y 319.734,Z 263.657,A -85,B 0,C 180,E1 -15133.992,E2 -15133.992} C_VEL
LIN {X 0,Y 319.661,Z 263.667,A -85,B 0,C 180,E1 -15137.927,E2 -15137.927} C_VEL
LIN {X 0,Y 319.606,Z 263.672,A -85,B 0,C 180,E1 -15140.6,E2 -15140.6} C_VEL
LIN {X 0,Y 319.544,Z 263.679,A -85,B 0,C 180,E1 -15143.321,E2 -15143.321} C_VEL
LIN {X 0,Y 319.555,Z 263.681,A -85,B 0,C 180,E1 -15146.095,E2 -15146.095} C_VEL
LIN {X 0,Y 319.545,Z 263.679,A -85,B 0,C 180,E1 -15148.938,E2 -15148.938} C_VEL
LIN {X 0,Y 319.527,Z 263.685,A -85,B 0,C 180,E1 -15151.862,E2 -15151.862} C_VEL
LIN {X 0,Y 319.582,Z 263.68,A -85,B 0,C 180,E1 -15155.543,E2 -15155.543} C_VEL
LIN {X 0,Y 319.529,Z 263.685,A -85,B 0,C 180,E1 -15159.662,E2 -15159.662} C_VEL
LIN {X 0,Y 319.522,Z 263.685,A -85,B 0,C 180,E1 -15163.46,E2 -15163.46} C_VEL
LIN {X 0,Y 319.55,Z 263.851,A -85,B 0,C 180,E1 -15165.011,E2 -15165.011} C_VEL
LIN {X 0,Y 320.398,Z 268.387,A -85,B 0,C 180,E1 -15168.848,E2 -15168.848} C_VEL
LIN {X 0,Y 321.024,Z 272.638,A -85,B 0,C 180,E1 -15172.194,E2 -15172.194} C_VEL
LIN {X 0,Y 321.066,Z 276.894,A -85,B 0,C 180,E1 -15175.31,E2 -15175.31} C_VEL
LIN {X 0,Y 320.333,Z 281.97,A -85,B 0,C 180,E1 -15178.831,E2 -15178.831} C_VEL
LIN {X 0,Y 319.642,Z 287.405,A -85,B 0,C 180,E1 -15182.501,E2 -15182.501} C_VEL
LIN {X 0,Y 319.121,Z 292.601,A -85,B 0,C 180,E1 -15185.957,E2 -15185.957} C_VEL
LIN {X 0,Y 319.009,Z 294.399,A -85,B 0,C 180,E1 -15187.126,E2 -15187.126} C_VEL
LIN {X 0,Y 322.006,Z 307.624,A -85,B 0,C 180,E1 -15187.887,E2 -15187.887} C_VEL
LIN {X 0,Y 324.134,Z 320.006,A -85,B 0,C 180,E1 -15188.803,E2 -15188.803} C_VEL
LIN {X 0,Y 325.333,Z 330.905,A -85,B 0,C 180,E1 -15189.779,E2 -15189.779} C_VEL
LIN {X 0,Y 325.608,Z 337.55,A -85,B 0,C 180,E1 -15190.454,E2 -15190.454} C_VEL
LIN {X 0,Y 324.172,Z 348.511,A -85,B 0,C 180,E1 -15191.678,E2 -15191.678} C_VEL
LIN {X 0,Y 322.933,Z 357.429,A -85,B 0,C 180,E1 -15192.914,E2 -15192.914} C_VEL
LIN {X 0,Y 321.607,Z 367.001,A -85,B 0,C 180,E1 -15194.554,E2 -15194.554} C_VEL
LIN {X 0,Y 320.422,Z 375.529,A -85,B 0,C 180,E1 -15196.362,E2 -15196.362} C_VEL
LIN {X 0,Y 319.325,Z 382.717,A -85,B 0,C 180,E1 -15198.253,E2 -15198.253} C_VEL
LIN {X 0,Y 318.736,Z 387.574,A -85,B 0,C 180,E1 -15199.84,E2 -15199.84} C_VEL
LIN {X 0,Y 318.212,Z 392.296,A -85,B 0,C 180,E1 -15201.746,E2 -15201.746} C_VEL
LIN {X 0,Y 317.908,Z 395.905,A -85,B 0,C 180,E1 -15203.654,E2 -15203.654} C_VEL
LIN {X 0,Y 317.81,Z 397.767,A -85,B 0,C 180,E1 -15204.925,E2 -15204.925} C_VEL
LIN {X 0,Y 317.808,Z 399.165,A -85,B 0,C 180,E1 -15206.196,E2 -15206.196} C_VEL
LIN {X 0,Y 317.758,Z 400.161,A -85,B 0,C 180,E1 -15207.465,E2 -15207.465} C_VEL
LIN {X 0,Y 317.743,Z 400.769,A -85,B 0,C 180,E1 -15208.732,E2 -15208.732} C_VEL
LIN {X 0,Y 317.781,Z 400.984,A -85,B 0,C 180,E1 -15210,E2 -15210} C_VEL
LIN {X 0,Y 317.743,Z 400.763,A -85,B 0,C 180,E1 -15211.267,E2 -15211.267} C_VEL
LIN {X 0,Y 317.757,Z 400.152,A -85,B 0,C 180,E1 -15212.535,E2 -15212.535} C_VEL
LIN {X 0,Y 317.802,Z 399.152,A -85,B 0,C 180,E1 -15213.804,E2 -15213.804} C_VEL
LIN {X 0,Y 317.826,Z 396.885,A -85,B 0,C 180,E1 -15215.688,E2 -15215.688} C_VEL
LIN {X 0,Y 318.076,Z 393.572,A -85,B 0,C 180,E1 -15217.618,E2 -15217.618} C_VEL
LIN {X 0,Y 318.545,Z 389.223,A -85,B 0,C 180,E1 -15219.525,E2 -15219.525} C_VEL
LIN {X 0,Y 319.2,Z 383.684,A -85,B 0,C 180,E1 -15221.429,E2 -15221.429} C_VEL
LIN {X 0,Y 320.217,Z 376.776,A -85,B 0,C 180,E1 -15223.323,E2 -15223.323} C_VEL
LIN {X 0,Y 321.238,Z 369.723,A -85,B 0,C 180,E1 -15224.896,E2 -15224.896} C_VEL
LIN {X 0,Y 322.407,Z 361.223,A -85,B 0,C 180,E1 -15226.462,E2 -15226.462} C_VEL
LIN {X 0,Y 323.852,Z 350.723,A -85,B 0,C 180,E1 -15228.014,E2 -15228.014} C_VEL
LIN {X 0,Y 325.217,Z 340.338,A -85,B 0,C 180,E1 -15229.242,E2 -15229.242} C_VEL
LIN {X 0,Y 325.561,Z 334.178,A -85,B 0,C 180,E1 -15229.877,E2 -15229.877} C_VEL
LIN {X 0,Y 324.592,Z 323.594,A -85,B 0,C 180,E1 -15230.878,E2 -15230.878} C_VEL
LIN {X 0,Y 322.526,Z 310.534,A -85,B 0,C 180,E1 -15231.894,E2 -15231.894} C_VEL
LIN {X 0,Y 319.852,Z 298.355,A -85,B 0,C 180,E1 -15232.653,E2 -15232.653} C_VEL
LIN {X 0,Y 318.996,Z 294.363,A -85,B 0,C 180,E1 -15232.858,E2 -15232.858} C_VEL
LIN {X 0,Y 319.551,Z 288.418,A -85,B 0,C 180,E1 -15236.799,E2 -15236.799} C_VEL
LIN {X 0,Y 320.157,Z 283.163,A -85,B 0,C 180,E1 -15240.324,E2 -15240.324} C_VEL
LIN {X 0,Y 320.85,Z 278.326,A -85,B 0,C 180,E1 -15243.657,E2 -15243.657} C_VEL
LIN {X 0,Y 321.088,Z 274.708,A -85,B 0,C 180,E1 -15246.226,E2 -15246.226} C_VEL
LIN {X 0,Y 320.996,Z 272.37,A -85,B 0,C 180,E1 -15247.982,E2 -15247.982} C_VEL
LIN {X 0,Y 320.385,Z 268.346,A -85,B 0,C 180,E1 -15251.154,E2 -15251.154} C_VEL
LIN {X 0,Y 319.518,Z 263.686,A -85,B 0,C 180,E1 -15255.124,E2 -15255.124} C_VEL
LIN {X 0,Y 319.5,Z 263.687,A -85,B 0,C 180,E1 -15258.707,E2 -15258.707} C_VEL
LIN {X 0,Y 319.547,Z 263.682,A -85,B 0,C 180,E1 -15262.351,E2 -15262.351} C_VEL
LIN {X 0,Y 319.561,Z 263.678,A -85,B 0,C 180,E1 -15265.123,E2 -15265.123} C_VEL
LIN {X 0,Y 319.526,Z 263.686,A -85,B 0,C 180,E1 -15268.137,E2 -15268.137} C_VEL
LIN {X 0,Y 319.572,Z 263.677,A -85,B 0,C 180,E1 -15271.603,E2 -15271.603} C_VEL
LIN {X 0,Y 319.549,Z 263.679,A -85,B 0,C 180,E1 -15275.299,E2 -15275.299} C_VEL
LIN {X 0,Y 319.566,Z 263.681,A -85,B 0,C 180,E1 -15278.046,E2 -15278.046} C_VEL
LIN {X 0,Y 319.69,Z 263.661,A -85,B 0,C 180,E1 -15280.962,E2 -15280.962} C_VEL
LIN {X 0,Y 319.732,Z 263.657,A -85,B 0,C 180,E1 -15285.276,E2 -15285.276} C_VEL
LIN {X 0,Y 319.716,Z 263.657,A -85,B 0,C 180,E1 -15288.589,E2 -15288.589} C_VEL
LIN {X 0,Y 319.895,Z 263.634,A -85,B 0,C 180,E1 -15292.425,E2 -15292.425} C_VEL
LIN {X 0,Y 319.744,Z 263.655,A -85,B 0,C 180,E1 -15294.956,E2 -15294.956} C_VEL
LIN {X 0,Y 319.991,Z 263.626,A -85,B 0,C 180,E1 -15297.482,E2 -15297.482} C_VEL
LIN {X 0,Y 320.113,Z 263.608,A -85,B 0,C 180,E1 -15300,E2 -15300} C_VEL
LIN {X 0,Y 319.961,Z 263.627,A -85,B 0,C 180,E1 -15302.518,E2 -15302.518} C_VEL
LIN {X 0,Y 319.897,Z 263.633,A -85,B 0,C 180,E1 -15306.606,E2 -15306.606} C_VEL
LIN {X 0,Y 319.737,Z 263.655,A -85,B 0,C 180,E1 -15310.128,E2 -15310.128} C_VEL
LIN {X 0,Y 319.734,Z 263.655,A -85,B 0,C 180,E1 -15313.992,E2 -15313.992} C_VEL
LIN {X 0,Y 319.625,Z 263.669,A -85,B 0,C 180,E1 -15317.929,E2 -15317.929} C_VEL
LIN {X 0,Y 319.569,Z 263.676,A -85,B 0,C 180,E1 -15321.954,E2 -15321.954} C_VEL
LIN {X 0,Y 319.636,Z 263.67,A -85,B 0,C 180,E1 -15326.088,E2 -15326.088} C_VEL
LIN {X 0,Y 319.599,Z 263.672,A -85,B 0,C 180,E1 -15328.933,E2 -15328.933} C_VEL
LIN {X 0,Y 319.533,Z 263.683,A -85,B 0,C 180,E1 -15331.862,E2 -15331.862} C_VEL
LIN {X 0,Y 319.579,Z 263.676,A -85,B 0,C 180,E1 -15335.543,E2 -15335.543} C_VEL
LIN {X 0,Y 319.573,Z 263.68,A -85,B 0,C 180,E1 -15338.008,E2 -15338.008} C_VEL
LIN {X 0,Y 319.525,Z 263.685,A -85,B 0,C 180,E1 -15341.597,E2 -15341.597} C_VEL
LIN {X 0,Y 319.487,Z 263.687,A -85,B 0,C 180,E1 -15345.257,E2 -15345.257} C_VEL
LIN {X 0,Y 319.504,Z 263.685,A -85,B 0,C 180,E1 -15348.408,E2 -15348.408} C_VEL
LIN {X 0,Y 319.5,Z 263.689,A -85,B 0,C 180,E1 -15351.982,E2 -15351.982} C_VEL
LIN {X 0,Y 319.503,Z 263.689,A -85,B 0,C 180,E1 -15352.362,E2 -15352.362} C_VEL
LIN {X 0,Y 319.556,Z 266.084,A -85,B 0,C 180,E1 -15355.123,E2 -15355.123} C_VEL
LIN {X 0,Y 319.373,Z 269.058,A -85,B 0,C 180,E1 -15358.121,E2 -15358.121} C_VEL
LIN {X 0,Y 319.12,Z 272.82,A -85,B 0,C 180,E1 -15361.754,E2 -15361.754} C_VEL
LIN {X 0,Y 318.815,Z 276.585,A -85,B 0,C 180,E1 -15365.239,E2 -15365.239} C_VEL
LIN {X 0,Y 318.684,Z 278.849,A -85,B 0,C 180,E1 -15367.198,E2 -15367.198} C_VEL
LIN {X 0,Y 322.438,Z 291.942,A -85,B 0,C 180,E1 -15368.048,E2 -15368.048} C_VEL
LIN {X 0,Y 325.094,Z 303.812,A -85,B 0,C 180,E1 -15368.998,E2 -15368.998} C_VEL
LIN {X 0,Y 326.72,Z 312.979,A -85,B 0,C 180,E1 -15369.869,E2 -15369.869} C_VEL
LIN {X 0,Y 326.727,Z 316.469,A -85,B 0,C 180,E1 -15370.197,E2 -15370.197} C_VEL
LIN {X 0,Y 325.38,Z 328.117,A -85,B 0,C 180,E1 -15371.423,E2 -15371.423} C_VEL
LIN {X 0,Y 324.04,Z 339.096,A -85,B 0,C 180,E1 -15372.893,E2 -15372.893} C_VEL
LIN {X 0,Y 322.701,Z 348.797,A -85,B 0,C 180,E1 -15374.527,E2 -15374.527} C_VEL
LIN {X 0,Y 321.231,Z 357.71,A -85,B 0,C 180,E1 -15376.397,E2 -15376.397} C_VEL
LIN {X 0,Y 320.163,Z 364.88,A -85,B 0,C 180,E1 -15378.285,E2 -15378.285} C_VEL
LIN {X 0,Y 319.417,Z 369.715,A -85,B 0,C 180,E1 -15379.862,E2 -15379.862} C_VEL
LIN {X 0,Y 318.753,Z 374.412,A -85,B 0,C 180,E1 -15381.76,E2 -15381.76} C_VEL
LIN {X 0,Y 318.336,Z 378.005,A -85,B 0,C 180,E1 -15383.663,E2 -15383.663} C_VEL
LIN {X 0,Y 318.157,Z 379.861,A -85,B 0,C 180,E1 -15384.931,E2 -15384.931} C_VEL
LIN {X 0,Y 317.988,Z 381.258,A -85,B 0,C 180,E1 -15386.198,E2 -15386.198} C_VEL
LIN {X 0,Y 317.786,Z 382.864,A -85,B 0,C 180,E1 -15388.733,E2 -15388.733} C_VEL
LIN {X 0,Y 317.787,Z 383.095,A -85,B 0,C 180,E1 -15390,E2 -15390} C_VEL
LIN {X 0,Y 317.786,Z 382.904,A -85,B 0,C 180,E1 -15391.267,E2 -15391.267} C_VEL
LIN {X 0,Y 317.985,Z 381.35,A -85,B 0,C 180,E1 -15393.802,E2 -15393.802} C_VEL
LIN {X 0,Y 318.151,Z 379.993,A -85,B 0,C 180,E1 -15395.069,E2 -15395.069} C_VEL
LIN {X 0,Y 318.398,Z 377.676,A -85,B 0,C 180,E1 -15396.642,E2 -15396.642} C_VEL
LIN {X 0,Y 318.927,Z 373.241,A -85,B 0,C 180,E1 -15398.874,E2 -15398.874} C_VEL
LIN {X 0,Y 319.679,Z 368.223,A -85,B 0,C 180,E1 -15400.77,E2 -15400.77} C_VEL
LIN {X 0,Y 320.654,Z 361.905,A -85,B 0,C 180,E1 -15402.661,E2 -15402.661} C_VEL
LIN {X 0,Y 321.848,Z 353.997,A -85,B 0,C 180,E1 -15404.544,E2 -15404.544} C_VEL
LIN {X 0,Y 323.401,Z 344.155,A -85,B 0,C 180,E1 -15406.41,E2 -15406.41} C_VEL
LIN {X 0,Y 324.719,Z 333.827,A -85,B 0,C 180,E1 -15407.964,E2 -15407.964} C_VEL
LIN {X 0,Y 325.96,Z 323.594,A -85,B 0,C 180,E1 -15409.196,E2 -15409.196} C_VEL
LIN {X 0,Y 326.87,Z 314.158,A -85,B 0,C 180,E1 -15410.122,E2 -15410.122} C_VEL
LIN {X 0,Y 324.826,Z 302.382,A -85,B 0,C 180,E1 -15411.238,E2 -15411.238} C_VEL
LIN {X 0,Y 321.993,Z 290.32,A -85,B 0,C 180,E1 -15412.187,E2 -15412.187} C_VEL
LIN {X 0,Y 318.682,Z 278.749,A -85,B 0,C 180,E1 -15412.93,E2 -15412.93} C_VEL
LIN {X 0,Y 318.909,Z 275.177,A -85,B 0,C 180,E1 -15416.152,E2 -15416.152} C_VEL
LIN {X 0,Y 319.142,Z 272.184,A -85,B 0,C 180,E1 -15418.978,E2 -15418.978} C_VEL
LIN {X 0,Y 319.352,Z 269.187,A -85,B 0,C 180,E1 -15421.882,E2 -15421.882} C_VEL
LIN {X 0,Y 319.551,Z 265.568,A -85,B 0,C 180,E1 -15425.535,E2 -15425.535} C_VEL
LIN {X 0,Y 319.496,Z 263.687,A -85,B 0,C 180,E1 -15427.636,E2 -15427.636} C_VEL
LIN {X 0,Y 319.5,Z 263.682,A -85,B 0,C 180,E1 -15431.293,E2 -15431.293} C_VEL
LIN {X 0,Y 319.521,Z 263.68,A -85,B 0,C 180,E1 -15433.46,E2 -15433.46} C_VEL
LIN {X 0,Y 319.555,Z 263.678,A -85,B 0,C 180,E1 -15437.016,E2 -15437.016} C_VEL
LIN {X 0,Y 319.549,Z 263.682,A -85,B 0,C 180,E1 -15440.371,E2 -15440.371} C_VEL
LIN {X 0,Y 319.561,Z 263.678,A -85,B 0,C 180,E1 -15443.572,E2 -15443.572} C_VEL
LIN {X 0,Y 319.579,Z 263.675,A -85,B 0,C 180,E1 -15446.687,E2 -15446.687} C_VEL
LIN {X 0,Y 319.594,Z 263.675,A -85,B 0,C 180,E1 -15449.617,E2 -15449.617} C_VEL
LIN {X 0,Y 319.611,Z 263.669,A -85,B 0,C 180,E1 -15452.498,E2 -15452.498} C_VEL
LIN {X 0,Y 319.635,Z 263.67,A -85,B 0,C 180,E1 -15454.08,E2 -15454.08} C_VEL
LIN {X 0,Y 318.959,Z 263.755,A -85,B 0,C 180,E1 -15455.132,E2 -15455.132} C_VEL
LIN {X 0,Y 316.065,Z 264.11,A -85,B 0,C 180,E1 -15456.843,E2 -15456.843} C_VEL
LIN {X 0,Y 313.625,Z 264.417,A -85,B 0,C 180,E1 -15458.23,E2 -15458.23} C_VEL
LIN {X 0,Y 312.598,Z 264.547,A -85,B 0,C 180,E1 -15459.305,E2 -15459.305} C_VEL
LIN {X 0,Y 312.525,Z 264.551,A -85,B 0,C 180,E1 -15459.669,E2 -15459.669} C_VEL
LIN {X 0,Y 312.583,Z 264.547,A -85,B 0,C 180,E1 -15463.005,E2 -15463.005} C_VEL
LIN {X 0,Y 312.688,Z 264.535,A -85,B 0,C 180,E1 -15465.686,E2 -15465.686} C_VEL
LIN {X 0,Y 312.688,Z 264.534,A -85,B 0,C 180,E1 -15469.641,E2 -15469.641} C_VEL
LIN {X 0,Y 312.822,Z 264.516,A -85,B 0,C 180,E1 -15472.253,E2 -15472.253} C_VEL
LIN {X 0,Y 312.7,Z 264.535,A -85,B 0,C 180,E1 -15474.842,E2 -15474.842} C_VEL
LIN {X 0,Y 312.971,Z 264.502,A -85,B 0,C 180,E1 -15478.713,E2 -15478.713} C_VEL
LIN {X 0,Y 312.938,Z 264.505,A -85,B 0,C 180,E1 -15482.574,E2 -15482.574} C_VEL
LIN {X 0,Y 312.895,Z 264.511,A -85,B 0,C 180,E1 -15486.448,E2 -15486.448} C_VEL
LIN {X 0,Y 312.686,Z 264.537,A -85,B 0,C 180,E1 -15490.359,E2 -15490.359} C_VEL
LIN {X 0,Y 312.703,Z 264.531,A -85,B 0,C 180,E1 -15494.888,E2 -15494.888} C_VEL
LIN {X 0,Y 312.632,Z 264.54,A -85,B 0,C 180,E1 -15499.236,E2 -15499.236} C_VEL
LIN {X 0,Y 312.52,Z 264.554,A -85,B 0,C 180,E1 -15502.777,E2 -15502.777} C_VEL
LIN {X 0,Y 312.489,Z 264.558,A -85,B 0,C 180,E1 -15506.731,E2 -15506.731} C_VEL
LIN {X 0,Y 312.498,Z 264.561,A -85,B 0,C 180,E1 -15509.655,E2 -15509.655} C_VEL
LIN {X 0,Y 312.522,Z 264.559,A -85,B 0,C 180,E1 -15513.689,E2 -15513.689} C_VEL
LIN {X 0,Y 312.516,Z 264.559,A -85,B 0,C 180,E1 -15517.387,E2 -15517.387} C_VEL
LIN {X 0,Y 312.442,Z 264.566,A -85,B 0,C 180,E1 -15520.717,E2 -15520.717} C_VEL
LIN {X 0,Y 312.484,Z 264.659,A -85,B 0,C 180,E1 -15524.542,E2 -15524.542} C_VEL
LIN {X 0,Y 313.373,Z 269.365,A -85,B 0,C 180,E1 -15528.622,E2 -15528.622} C_VEL
LIN {X 0,Y 313.905,Z 272.992,A -85,B 0,C 180,E1 -15531.593,E2 -15531.593} C_VEL
LIN {X 0,Y 314.087,Z 275.696,A -85,B 0,C 180,E1 -15533.662,E2 -15533.662} C_VEL
LIN {X 0,Y 313.905,Z 278.835,A -85,B 0,C 180,E1 -15535.963,E2 -15535.963} C_VEL
LIN {X 0,Y 313.118,Z 284.077,A -85,B 0,C 180,E1 -15539.667,E2 -15539.667} C_VEL
LIN {X 0,Y 312.475,Z 289.305,A -85,B 0,C 180,E1 -15543.267,E2 -15543.267} C_VEL
LIN {X 0,Y 311.983,Z 294.143,A -85,B 0,C 180,E1 -15546.57,E2 -15546.57} C_VEL
LIN {X 0,Y 315.207,Z 308.189,A -85,B 0,C 180,E1 -15547.427,E2 -15547.427} C_VEL
LIN {X 0,Y 317.403,Z 321.132,A -85,B 0,C 180,E1 -15548.431,E2 -15548.431} C_VEL
LIN {X 0,Y 318.614,Z 332.482,A -85,B 0,C 180,E1 -15549.502,E2 -15549.502} C_VEL
LIN {X 0,Y 318.736,Z 338.884,A -85,B 0,C 180,E1 -15550.183,E2 -15550.183} C_VEL
LIN {X 0,Y 317.247,Z 349.491,A -85,B 0,C 180,E1 -15551.431,E2 -15551.431} C_VEL
LIN {X 0,Y 315.824,Z 359.188,A -85,B 0,C 180,E1 -15552.851,E2 -15552.851} C_VEL
LIN {X 0,Y 314.557,Z 368.029,A -85,B 0,C 180,E1 -15554.448,E2 -15554.448} C_VEL
LIN {X 0,Y 313.513,Z 375.331,A -85,B 0,C 180,E1 -15556.055,E2 -15556.055} C_VEL
LIN {X 0,Y 312.344,Z 382.518,A -85,B 0,C 180,E1 -15557.987,E2 -15557.987} C_VEL
LIN {X 0,Y 311.709,Z 387.375,A -85,B 0,C 180,E1 -15559.608,E2 -15559.608} C_VEL
LIN {X 0,Y 311.154,Z 392.096,A -85,B 0,C 180,E1 -15561.557,E2 -15561.557} C_VEL
LIN {X 0,Y 310.832,Z 395.705,A -85,B 0,C 180,E1 -15563.509,E2 -15563.509} C_VEL
LIN {X 0,Y 310.713,Z 397.567,A -85,B 0,C 180,E1 -15564.809,E2 -15564.809} C_VEL
LIN {X 0,Y 310.719,Z 398.966,A -85,B 0,C 180,E1 -15566.109,E2 -15566.109} C_VEL
LIN {X 0,Y 310.682,Z 399.962,A -85,B 0,C 180,E1 -15567.407,E2 -15567.407} C_VEL
LIN {X 0,Y 310.657,Z 400.57,A -85,B 0,C 180,E1 -15568.704,E2 -15568.704} C_VEL
LIN {X 0,Y 310.692,Z 400.785,A -85,B 0,C 180,E1 -15570,E2 -15570} C_VEL
LIN {X 0,Y 310.657,Z 400.563,A -85,B 0,C 180,E1 -15571.296,E2 -15571.296} C_VEL
LIN {X 0,Y 310.681,Z 399.952,A -85,B 0,C 180,E1 -15572.593,E2 -15572.593} C_VEL
LIN {X 0,Y 310.712,Z 398.952,A -85,B 0,C 180,E1 -15573.891,E2 -15573.891} C_VEL
LIN {X 0,Y 310.723,Z 396.967,A -85,B 0,C 180,E1 -15575.614,E2 -15575.614} C_VEL
LIN {X 0,Y 311.018,Z 393.37,A -85,B 0,C 180,E1 -15577.792,E2 -15577.792} C_VEL
LIN {X 0,Y 311.499,Z 389.02,A -85,B 0,C 180,E1 -15579.742,E2 -15579.742} C_VEL
LIN {X 0,Y 312.19,Z 383.481,A -85,B 0,C 180,E1 -15581.689,E2 -15581.689} C_VEL
LIN {X 0,Y 313.274,Z 376.573,A -85,B 0,C 180,E1 -15583.624,E2 -15583.624} C_VEL
LIN {X 0,Y 314.338,Z 369.52,A -85,B 0,C 180,E1 -15585.231,E2 -15585.231} C_VEL
LIN {X 0,Y 315.568,Z 361.019,A -85,B 0,C 180,E1 -15586.829,E2 -15586.829} C_VEL
LIN {X 0,Y 317.093,Z 350.52,A -85,B 0,C 180,E1 -15588.411,E2 -15588.411} C_VEL
LIN {X 0,Y 318.685,Z 338.703,A -85,B 0,C 180,E1 -15589.82,E2 -15589.82} C_VEL
LIN {X 0,Y 318.559,Z 332.255,A -85,B 0,C 180,E1 -15590.501,E2 -15590.501} C_VEL
LIN {X 0,Y 317.355,Z 321.155,A -85,B 0,C 180,E1 -15591.547,E2 -15591.547} C_VEL
LIN {X 0,Y 315.154,Z 307.94,A -85,B 0,C 180,E1 -15592.567,E2 -15592.567} C_VEL
LIN {X 0,Y 312.067,Z 294.796,A -85,B 0,C 180,E1 -15593.371,E2 -15593.371} C_VEL
LIN {X 0,Y 311.991,Z 294.126,A -85,B 0,C 180,E1 -15593.419,E2 -15593.419} C_VEL
LIN {X 0,Y 312.581,Z 288.226,A -85,B 0,C 180,E1 -15597.446,E2 -15597.446} C_VEL
LIN {X 0,Y 313.385,Z 282.291,A -85,B 0,C 180,E1 -15601.549,E2 -15601.549} C_VEL
LIN {X 0,Y 314.044,Z 277.734,A -85,B 0,C 180,E1 -15604.796,E2 -15604.796} C_VEL
LIN {X 0,Y 314.073,Z 274.559,A -85,B 0,C 180,E1 -15607.17,E2 -15607.17} C_VEL
LIN {X 0,Y 313.503,Z 270.316,A -85,B 0,C 180,E1 -15610.55,E2 -15610.55} C_VEL
LIN {X 0,Y 312.743,Z 266.06,A -85,B 0,C 180,E1 -15614.158,E2 -15614.158} C_VEL
LIN {X 0,Y 312.456,Z 264.566,A -85,B 0,C 180,E1 -15615.566,E2 -15615.566} C_VEL
LIN {X 0,Y 312.441,Z 264.567,A -85,B 0,C 180,E1 -15619.283,E2 -15619.283} C_VEL
LIN {X 0,Y 312.515,Z 264.558,A -85,B 0,C 180,E1 -15622.613,E2 -15622.613} C_VEL
LIN {X 0,Y 312.52,Z 264.559,A -85,B 0,C 180,E1 -15626.311,E2 -15626.311} C_VEL
LIN {X 0,Y 312.497,Z 264.563,A -85,B 0,C 180,E1 -15630.345,E2 -15630.345} C_VEL
LIN {X 0,Y 312.511,Z 264.561,A -85,B 0,C 180,E1 -15634.099,E2 -15634.099} C_VEL
LIN {X 0,Y 312.54,Z 264.553,A -85,B 0,C 180,E1 -15637.525,E2 -15637.525} C_VEL
LIN {X 0,Y 312.64,Z 264.542,A -85,B 0,C 180,E1 -15641.656,E2 -15641.656} C_VEL
LIN {X 0,Y 312.695,Z 264.537,A -85,B 0,C 180,E1 -15645.686,E2 -15645.686} C_VEL
LIN {X 0,Y 312.686,Z 264.537,A -85,B 0,C 180,E1 -15649.641,E2 -15649.641} C_VEL
LIN {X 0,Y 312.893,Z 264.511,A -85,B 0,C 180,E1 -15653.552,E2 -15653.552} C_VEL
LIN {X 0,Y 312.937,Z 264.505,A -85,B 0,C 180,E1 -15657.426,E2 -15657.426} C_VEL
LIN {X 0,Y 313.067,Z 264.486,A -85,B 0,C 180,E1 -15660,E2 -15660} C_VEL
LIN {X 0,Y 312.91,Z 264.506,A -85,B 0,C 180,E1 -15662.575,E2 -15662.575} C_VEL
LIN {X 0,Y 312.864,Z 264.511,A -85,B 0,C 180,E1 -15666.587,E2 -15666.587} C_VEL
LIN {X 0,Y 312.687,Z 264.534,A -85,B 0,C 180,E1 -15670.359,E2 -15670.359} C_VEL
LIN {X 0,Y 312.669,Z 264.539,A -85,B 0,C 180,E1 -15674.865,E2 -15674.865} C_VEL
LIN {X 0,Y 312.587,Z 264.546,A -85,B 0,C 180,E1 -15679.213,E2 -15679.213} C_VEL
LIN {X 0,Y 312.527,Z 264.555,A -85,B 0,C 180,E1 -15682.781,E2 -15682.781} C_VEL
LIN {X 0,Y 312.604,Z 264.545,A -85,B 0,C 180,E1 -15685.936,E2 -15685.936} C_VEL
LIN {X 0,Y 312.55,Z 264.55,A -85,B 0,C 180,E1 -15689.65,E2 -15689.65} C_VEL
LIN {X 0,Y 312.52,Z 264.556,A -85,B 0,C 180,E1 -15693.689,E2 -15693.689} C_VEL
LIN {X 0,Y 312.526,Z 264.554,A -85,B 0,C 180,E1 -15697.385,E2 -15697.385} C_VEL
LIN {X 0,Y 312.49,Z 264.558,A -85,B 0,C 180,E1 -15700.709,E2 -15700.709} C_VEL
LIN {X 0,Y 312.451,Z 264.563,A -85,B 0,C 180,E1 -15704.21,E2 -15704.21} C_VEL
LIN {X 0,Y 312.455,Z 264.566,A -85,B 0,C 180,E1 -15707.925,E2 -15707.925} C_VEL
LIN {X 0,Y 312.455,Z 264.567,A -85,B 0,C 180,E1 -15711.93,E2 -15711.93} C_VEL
LIN {X 0,Y 312.482,Z 264.776,A -85,B 0,C 180,E1 -15712.609,E2 -15712.609} C_VEL
LIN {X 0,Y 312.556,Z 266.257,A -85,B 0,C 180,E1 -15714.224,E2 -15714.224} C_VEL
LIN {X 0,Y 312.397,Z 269.24,A -85,B 0,C 180,E1 -15717.321,E2 -15717.321} C_VEL
LIN {X 0,Y 312.178,Z 272.242,A -85,B 0,C 180,E1 -15720.312,E2 -15720.312} C_VEL
LIN {X 0,Y 311.873,Z 276.448,A -85,B 0,C 180,E1 -15724.342,E2 -15724.342} C_VEL
LIN {X 0,Y 311.646,Z 278.935,A -85,B 0,C 180,E1 -15726.616,E2 -15726.616} C_VEL
LIN {X 0,Y 316.179,Z 294.92,A -85,B 0,C 180,E1 -15727.748,E2 -15727.748} C_VEL
LIN {X 0,Y 318.774,Z 307.181,A -85,B 0,C 180,E1 -15728.809,E2 -15728.809} C_VEL
LIN {X 0,Y 320.052,Z 314.942,A -85,B 0,C 180,E1 -15729.598,E2 -15729.598} C_VEL
LIN {X 0,Y 319.01,Z 325.685,A -85,B 0,C 180,E1 -15730.703,E2 -15730.703} C_VEL
LIN {X 0,Y 317.731,Z 335.921,A -85,B 0,C 180,E1 -15732.015,E2 -15732.015} C_VEL
LIN {X 0,Y 316.344,Z 345.534,A -85,B 0,C 180,E1 -15733.545,E2 -15733.545} C_VEL
LIN {X 0,Y 314.839,Z 355.175,A -85,B 0,C 180,E1 -15735.456,E2 -15735.456} C_VEL
LIN {X 0,Y 313.561,Z 362.862,A -85,B 0,C 180,E1 -15737.377,E2 -15737.377} C_VEL
LIN {X 0,Y 312.438,Z 369.916,A -85,B 0,C 180,E1 -15739.633,E2 -15739.633} C_VEL
LIN {X 0,Y 311.71,Z 374.614,A -85,B 0,C 180,E1 -15741.573,E2 -15741.573} C_VEL
LIN {X 0,Y 311.267,Z 378.206,A -85,B 0,C 180,E1 -15743.518,E2 -15743.518} C_VEL
LIN {X 0,Y 311.09,Z 380.061,A -85,B 0,C 180,E1 -15744.815,E2 -15744.815} C_VEL
LIN {X 0,Y 310.925,Z 381.458,A -85,B 0,C 180,E1 -15746.112,E2 -15746.112} C_VEL
LIN {X 0,Y 310.7,Z 383.063,A -85,B 0,C 180,E1 -15748.704,E2 -15748.704} C_VEL
LIN {X 0,Y 310.698,Z 383.294,A -85,B 0,C 180,E1 -15750,E2 -15750} C_VEL
LIN {X 0,Y 310.7,Z 383.103,A -85,B 0,C 180,E1 -15751.296,E2 -15751.296} C_VEL
LIN {X 0,Y 310.922,Z 381.549,A -85,B 0,C 180,E1 -15753.888,E2 -15753.888} C_VEL
LIN {X 0,Y 311.084,Z 380.192,A -85,B 0,C 180,E1 -15755.185,E2 -15755.185} C_VEL
LIN {X 0,Y 311.437,Z 377.327,A -85,B 0,C 180,E1 -15757.129,E2 -15757.129} C_VEL
LIN {X 0,Y 311.922,Z 373.439,A -85,B 0,C 180,E1 -15759.075,E2 -15759.075} C_VEL
LIN {X 0,Y 312.701,Z 368.422,A -85,B 0,C 180,E1 -15761.014,E2 -15761.014} C_VEL
LIN {X 0,Y 313.722,Z 362.103,A -85,B 0,C 180,E1 -15762.945,E2 -15762.945} C_VEL
LIN {X 0,Y 314.985,Z 354.194,A -85,B 0,C 180,E1 -15764.868,E2 -15764.868} C_VEL
LIN {X 0,Y 316.589,Z 344.352,A -85,B 0,C 180,E1 -15766.774,E2 -15766.774} C_VEL
LIN {X 0,Y 317.812,Z 335.192,A -85,B 0,C 180,E1 -15768.201,E2 -15768.201} C_VEL
LIN {X 0,Y 319.097,Z 325.211,A -85,B 0,C 180,E1 -15769.459,E2 -15769.459} C_VEL
LIN {X 0,Y 320.138,Z 316.109,A -85,B 0,C 180,E1 -15770.396,E2 -15770.396} C_VEL
LIN {X 0,Y 318.438,Z 305.263,A -85,B 0,C 180,E1 -15771.482,E2 -15771.482} C_VEL
LIN {X 0,Y 315.64,Z 292.826,A -85,B 0,C 180,E1 -15772.527,E2 -15772.527} C_VEL
LIN {X 0,Y 312.013,Z 280.693,A -85,B 0,C 180,E1 -15773.374,E2 -15773.374} C_VEL
LIN {X 0,Y 311.65,Z 278.958,A -85,B 0,C 180,E1 -15773.479,E2 -15773.479} C_VEL
LIN {X 0,Y 311.916,Z 275.371,A -85,B 0,C 180,E1 -15776.785,E2 -15776.785} C_VEL
LIN {X 0,Y 312.14,Z 272.372,A -85,B 0,C 180,E1 -15779.693,E2 -15779.693} C_VEL
LIN {X 0,Y 312.366,Z 269.37,A -85,B 0,C 180,E1 -15782.683,E2 -15782.683} C_VEL
LIN {X 0,Y 312.533,Z 266.224,A -85,B 0,C 180,E1 -15785.949,E2 -15785.949} C_VEL
LIN {X 0,Y 312.451,Z 264.565,A -85,B 0,C 180,E1 -15788.069,E2 -15788.069} C_VEL
LIN {X 0,Y 312.457,Z 264.561,A -85,B 0,C 180,E1 -15792.075,E2 -15792.075} C_VEL
LIN {X 0,Y 312.459,Z 264.563,A -85,B 0,C 180,E1 -15796.035,E2 -15796.035} C_VEL
LIN {X 0,Y 312.506,Z 264.558,A -85,B 0,C 180,E1 -15799.875,E2 -15799.875} C_VEL
LIN {X 0,Y 312.539,Z 264.552,A -85,B 0,C 180,E1 -15802.617,E2 -15802.617} C_VEL
LIN {X 0,Y 312.522,Z 264.556,A -85,B 0,C 180,E1 -15806.311,E2 -15806.311} C_VEL
LIN {X 0,Y 312.548,Z 264.552,A -85,B 0,C 180,E1 -15810.35,E2 -15810.35} C_VEL
LIN {X 0,Y 312.605,Z 264.545,A -85,B 0,C 180,E1 -15814.067,E2 -15814.067} C_VEL
LIN {X 0,Y 312.567,Z 264.551,A -85,B 0,C 180,E1 -15817.527,E2 -15817.527} C_VEL
LIN {X 0,Y 312.525,Z 264.551,A -85,B 0,C 180,E1 -15819.669,E2 -15819.669} C_VEL
LIN {X 0,Y 311.914,Z 264.63,A -85,B 0,C 180,E1 -15820.744,E2 -15820.744} C_VEL
LIN {X 0,Y 309.171,Z 264.98,A -85,B 0,C 180,E1 -15822.496,E2 -15822.496} C_VEL
LIN {X 0,Y 306.797,Z 265.278,A -85,B 0,C 180,E1 -15823.917,E2 -15823.917} C_VEL
LIN {X 0,Y 305.734,Z 265.406,A -85,B 0,C 180,E1 -15825.015,E2 -15825.015} C_VEL
LIN {X 0,Y 305.625,Z 265.416,A -85,B 0,C 180,E1 -15825.387,E2 -15825.387} C_VEL
LIN {X 0,Y 305.628,Z 265.415,A -85,B 0,C 180,E1 -15829.399,E2 -15829.399} C_VEL
LIN {X 0,Y 305.768,Z 265.395,A -85,B 0,C 180,E1 -15832.073,E2 -15832.073} C_VEL
LIN {X 0,Y 305.67,Z 265.409,A -85,B 0,C 180,E1 -15834.723,E2 -15834.723} C_VEL
LIN {X 0,Y 305.939,Z 265.377,A -85,B 0,C 180,E1 -15838.684,E2 -15838.684} C_VEL
LIN {X 0,Y 305.957,Z 265.372,A -85,B 0,C 180,E1 -15841.316,E2 -15841.316} C_VEL
LIN {X 0,Y 305.686,Z 265.406,A -85,B 0,C 180,E1 -15845.277,E2 -15845.277} C_VEL
LIN {X 0,Y 305.774,Z 265.394,A -85,B 0,C 180,E1 -15847.927,E2 -15847.927} C_VEL
LIN {X 0,Y 305.599,Z 265.418,A -85,B 0,C 180,E1 -15851.945,E2 -15851.945} C_VEL
LIN {X 0,Y 305.64,Z 265.411,A -85,B 0,C 180,E1 -15855.035,E2 -15855.035} C_VEL
LIN {X 0,Y 305.578,Z 265.419,A -85,B 0,C 180,E1 -15859.444,E2 -15859.444} C_VEL
LIN {X 0,Y 305.473,Z 265.432,A -85,B 0,C 180,E1 -15863.032,E2 -15863.032} C_VEL
LIN {X 0,Y 305.456,Z 265.436,A -85,B 0,C 180,E1 -15866.191,E2 -15866.191} C_VEL
LIN {X 0,Y 305.451,Z 265.435,A -85,B 0,C 180,E1 -15869.034,E2 -15869.034} C_VEL
LIN {X 0,Y 305.439,Z 265.44,A -85,B 0,C 180,E1 -15871.953,E2 -15871.953} C_VEL
LIN {X 0,Y 305.464,Z 265.436,A -85,B 0,C 180,E1 -15875.113,E2 -15875.113} C_VEL
LIN {X 0,Y 305.435,Z 265.438,A -85,B 0,C 180,E1 -15878.525,E2 -15878.525} C_VEL
LIN {X 0,Y 305.437,Z 265.438,A -85,B 0,C 180,E1 -15882.582,E2 -15882.582} C_VEL
LIN {X 0,Y 305.431,Z 265.51,A -85,B 0,C 180,E1 -15884.088,E2 -15884.088} C_VEL
LIN {X 0,Y 306.299,Z 270.176,A -85,B 0,C 180,E1 -15888.287,E2 -15888.287} C_VEL
LIN {X 0,Y 306.925,Z 274.421,A -85,B 0,C 180,E1 -15891.811,E2 -15891.811} C_VEL
LIN {X 0,Y 307.047,Z 277.599,A -85,B 0,C 180,E1 -15894.291,E2 -15894.291} C_VEL
LIN {X 0,Y 306.711,Z 280.757,A -85,B 0,C 180,E1 -15896.637,E2 -15896.637} C_VEL
LIN {X 0,Y 306.066,Z 284.936,A -85,B 0,C 180,E1 -15899.657,E2 -15899.657} C_VEL
LIN {X 0,Y 305.322,Z 290.885,A -85,B 0,C 180,E1 -15903.859,E2 -15903.859} C_VEL
LIN {X 0,Y 304.999,Z 293.945,A -85,B 0,C 180,E1 -15905.999,E2 -15905.999} C_VEL
LIN {X 0,Y 308.271,Z 307.986,A -85,B 0,C 180,E1 -15906.89,E2 -15906.89} C_VEL
LIN {X 0,Y 310.531,Z 321.092,A -85,B 0,C 180,E1 -15907.941,E2 -15907.941} C_VEL
LIN {X 0,Y 311.772,Z 332.281,A -85,B 0,C 180,E1 -15909.031,E2 -15909.031} C_VEL
LIN {X 0,Y 312.034,Z 338.688,A -85,B 0,C 180,E1 -15909.739,E2 -15909.739} C_VEL
LIN {X 0,Y 310.326,Z 350.471,A -85,B 0,C 180,E1 -15911.172,E2 -15911.172} C_VEL
LIN {X 0,Y 308.729,Z 360.938,A -85,B 0,C 180,E1 -15912.786,E2 -15912.786} C_VEL
LIN {X 0,Y 307.444,Z 369.413,A -85,B 0,C 180,E1 -15914.419,E2 -15914.419} C_VEL
LIN {X 0,Y 306.18,Z 377.688,A -85,B 0,C 180,E1 -15916.392,E2 -15916.392} C_VEL
LIN {X 0,Y 305.079,Z 384.356,A -85,B 0,C 180,E1 -15918.371,E2 -15918.371} C_VEL
LIN {X 0,Y 304.289,Z 390.463,A -85,B 0,C 180,E1 -15920.696,E2 -15920.696} C_VEL
LIN {X 0,Y 303.842,Z 394.433,A -85,B 0,C 180,E1 -15922.691,E2 -15922.691} C_VEL
LIN {X 0,Y 303.638,Z 397.368,A -85,B 0,C 180,E1 -15924.688,E2 -15924.688} C_VEL
LIN {X 0,Y 303.632,Z 398.766,A -85,B 0,C 180,E1 -15926.018,E2 -15926.018} C_VEL
LIN {X 0,Y 303.607,Z 399.763,A -85,B 0,C 180,E1 -15927.346,E2 -15927.346} C_VEL
LIN {X 0,Y 303.574,Z 400.371,A -85,B 0,C 180,E1 -15928.673,E2 -15928.673} C_VEL
LIN {X 0,Y 303.604,Z 400.585,A -85,B 0,C 180,E1 -15930,E2 -15930} C_VEL
LIN {X 0,Y 303.574,Z 400.364,A -85,B 0,C 180,E1 -15931.326,E2 -15931.326} C_VEL
LIN {X 0,Y 303.605,Z 399.753,A -85,B 0,C 180,E1 -15932.653,E2 -15932.653} C_VEL
LIN {X 0,Y 303.606,Z 398.751,A -85,B 0,C 180,E1 -15933.982,E2 -15933.982} C_VEL
LIN {X 0,Y 303.618,Z 397.058,A -85,B 0,C 180,E1 -15935.53,E2 -15935.53} C_VEL
LIN {X 0,Y 303.957,Z 393.169,A -85,B 0,C 180,E1 -15937.974,E2 -15937.974} C_VEL
LIN {X 0,Y 304.462,Z 388.818,A -85,B 0,C 180,E1 -15939.969,E2 -15939.969} C_VEL
LIN {X 0,Y 305.195,Z 383.278,A -85,B 0,C 180,E1 -15941.961,E2 -15941.961} C_VEL
LIN {X 0,Y 306.354,Z 376.371,A -85,B 0,C 180,E1 -15943.938,E2 -15943.938} C_VEL
LIN {X 0,Y 307.468,Z 369.317,A -85,B 0,C 180,E1 -15945.58,E2 -15945.58} C_VEL
LIN {X 0,Y 308.745,Z 360.815,A -85,B 0,C 180,E1 -15947.213,E2 -15947.213} C_VEL
LIN {X 0,Y 310.315,Z 350.315,A -85,B 0,C 180,E1 -15948.828,E2 -15948.828} C_VEL
LIN {X 0,Y 311.97,Z 338.498,A -85,B 0,C 180,E1 -15950.265,E2 -15950.265} C_VEL
LIN {X 0,Y 311.336,Z 328.093,A -85,B 0,C 180,E1 -15951.383,E2 -15951.383} C_VEL
LIN {X 0,Y 309.751,Z 316.185,A -85,B 0,C 180,E1 -15952.457,E2 -15952.457} C_VEL
LIN {X 0,Y 307.352,Z 303.802,A -85,B 0,C 180,E1 -15953.373,E2 -15953.373} C_VEL
LIN {X 0,Y 304.98,Z 293.96,A -85,B 0,C 180,E1 -15953.966,E2 -15953.966} C_VEL
LIN {X 0,Y 305.643,Z 288.031,A -85,B 0,C 180,E1 -15958.124,E2 -15958.124} C_VEL
LIN {X 0,Y 306.385,Z 282.678,A -85,B 0,C 180,E1 -15961.927,E2 -15961.927} C_VEL
LIN {X 0,Y 307.028,Z 278.62,A -85,B 0,C 180,E1 -15964.908,E2 -15964.908} C_VEL
LIN {X 0,Y 307.052,Z 276.181,A -85,B 0,C 180,E1 -15966.764,E2 -15966.764} C_VEL
LIN {X 0,Y 306.623,Z 272.274,A -85,B 0,C 180,E1 -15969.924,E2 -15969.924} C_VEL
LIN {X 0,Y 305.882,Z 268.008,A -85,B 0,C 180,E1 -15973.574,E2 -15973.574} C_VEL
LIN {X 0,Y 305.416,Z 265.442,A -85,B 0,C 180,E1 -15976.128,E2 -15976.128} C_VEL
LIN {X 0,Y 305.41,Z 265.443,A -85,B 0,C 180,E1 -15979.885,E2 -15979.885} C_VEL
LIN {X 0,Y 305.464,Z 265.434,A -85,B 0,C 180,E1 -15983.636,E2 -15983.636} C_VEL
LIN {X 0,Y 305.466,Z 265.438,A -85,B 0,C 180,E1 -15986.483,E2 -15986.483} C_VEL
LIN {X 0,Y 305.431,Z 265.439,A -85,B 0,C 180,E1 -15989.587,E2 -15989.587} C_VEL
LIN {X 0,Y 305.453,Z 265.438,A -85,B 0,C 180,E1 -15992.602,E2 -15992.602} C_VEL
LIN {X 0,Y 305.459,Z 265.436,A -85,B 0,C 180,E1 -15995.535,E2 -15995.535} C_VEL
LIN {X 0,Y 305.507,Z 265.432,A -85,B 0,C 180,E1 -15999.814,E2 -15999.814} C_VEL
LIN {X 0,Y 305.576,Z 265.419,A -85,B 0,C 180,E1 -16002.603,E2 -16002.603} C_VEL
LIN {X 0,Y 305.65,Z 265.411,A -85,B 0,C 180,E1 -16005.349,E2 -16005.349} C_VEL
LIN {X 0,Y 305.625,Z 265.416,A -85,B 0,C 180,E1 -16009.399,E2 -16009.399} C_VEL
LIN {X 0,Y 305.773,Z 265.395,A -85,B 0,C 180,E1 -16012.073,E2 -16012.073} C_VEL
LIN {X 0,Y 305.685,Z 265.405,A -85,B 0,C 180,E1 -16014.723,E2 -16014.723} C_VEL
LIN {X 0,Y 305.957,Z 265.371,A -85,B 0,C 180,E1 -16018.684,E2 -16018.684} C_VEL
LIN {X 0,Y 305.949,Z 265.376,A -85,B 0,C 180,E1 -16021.316,E2 -16021.316} C_VEL
LIN {X 0,Y 305.819,Z 265.39,A -85,B 0,C 180,E1 -16026.598,E2 -16026.598} C_VEL
LIN {X 0,Y 305.695,Z 265.406,A -85,B 0,C 180,E1 -16029.261,E2 -16029.261} C_VEL
LIN {X 0,Y 305.589,Z 265.418,A -85,B 0,C 180,E1 -16033.296,E2 -16033.296} C_VEL
LIN {X 0,Y 305.553,Z 265.422,A -85,B 0,C 180,E1 -16036.022,E2 -16036.022} C_VEL
LIN {X 0,Y 305.543,Z 265.423,A -85,B 0,C 180,E1 -16039.427,E2 -16039.427} C_VEL
LIN {X 0,Y 305.487,Z 265.431,A -85,B 0,C 180,E1 -16043.039,E2 -16043.039} C_VEL
LIN {X 0,Y 305.549,Z 265.426,A -85,B 0,C 180,E1 -16046.227,E2 -16046.227} C_VEL
LIN {X 0,Y 305.504,Z 265.427,A -85,B 0,C 180,E1 -16049.052,E2 -16049.052} C_VEL
LIN {X 0,Y 305.466,Z 265.434,A -85,B 0,C 180,E1 -16053.517,E2 -16053.517} C_VEL
LIN {X 0,Y 305.475,Z 265.432,A -85,B 0,C 180,E1 -16056.74,E2 -16056.74} C_VEL
LIN {X 0,Y 305.455,Z 265.435,A -85,B 0,C 180,E1 -16060.6,E2 -16060.6} C_VEL
LIN {X 0,Y 305.426,Z 265.442,A -85,B 0,C 180,E1 -16063.655,E2 -16063.655} C_VEL
LIN {X 0,Y 305.435,Z 265.44,A -85,B 0,C 180,E1 -16067.419,E2 -16067.419} C_VEL
LIN {X 0,Y 305.403,Z 265.445,A -85,B 0,C 180,E1 -16071.587,E2 -16071.587} C_VEL
LIN {X 0,Y 305.506,Z 266.764,A -85,B 0,C 180,E1 -16073.626,E2 -16073.626} C_VEL
LIN {X 0,Y 305.427,Z 269.425,A -85,B 0,C 180,E1 -16076.479,E2 -16076.479} C_VEL
LIN {X 0,Y 305.183,Z 272.426,A -85,B 0,C 180,E1 -16079.56,E2 -16079.56} C_VEL
LIN {X 0,Y 304.925,Z 275.442,A -85,B 0,C 180,E1 -16082.551,E2 -16082.551} C_VEL
LIN {X 0,Y 304.635,Z 279.157,A -85,B 0,C 180,E1 -16086.074,E2 -16086.074} C_VEL
LIN {X 0,Y 308.492,Z 292.34,A -85,B 0,C 180,E1 -16086.997,E2 -16086.997} C_VEL
LIN {X 0,Y 311.352,Z 304.594,A -85,B 0,C 180,E1 -16088.051,E2 -16088.051} C_VEL
LIN {X 0,Y 313.2,Z 315.154,A -85,B 0,C 180,E1 -16089.132,E2 -16089.132} C_VEL
LIN {X 0,Y 313.238,Z 318.463,A -85,B 0,C 180,E1 -16089.478,E2 -16089.478} C_VEL
LIN {X 0,Y 311.797,Z 329.81,A -85,B 0,C 180,E1 -16090.752,E2 -16090.752} C_VEL
LIN {X 0,Y 310.459,Z 339.506,A -85,B 0,C 180,E1 -16092.12,E2 -16092.12} C_VEL
LIN {X 0,Y 309.034,Z 349.202,A -85,B 0,C 180,E1 -16093.824,E2 -16093.824} C_VEL
LIN {X 0,Y 307.444,Z 358.114,A -85,B 0,C 180,E1 -16095.775,E2 -16095.775} C_VEL
LIN {X 0,Y 306.252,Z 365.284,A -85,B 0,C 180,E1 -16097.745,E2 -16097.745} C_VEL
LIN {X 0,Y 305.439,Z 370.118,A -85,B 0,C 180,E1 -16099.393,E2 -16099.393} C_VEL
LIN {X 0,Y 304.695,Z 374.815,A -85,B 0,C 180,E1 -16101.377,E2 -16101.377} C_VEL
LIN {X 0,Y 304.195,Z 378.529,A -85,B 0,C 180,E1 -16103.443,E2 -16103.443} C_VEL
LIN {X 0,Y 304.024,Z 380.262,A -85,B 0,C 180,E1 -16104.695,E2 -16104.695} C_VEL
LIN {X 0,Y 303.864,Z 381.657,A -85,B 0,C 180,E1 -16106.021,E2 -16106.021} C_VEL
LIN {X 0,Y 303.616,Z 383.263,A -85,B 0,C 180,E1 -16108.674,E2 -16108.674} C_VEL
LIN {X 0,Y 303.61,Z 383.494,A -85,B 0,C 180,E1 -16110,E2 -16110} C_VEL
LIN {X 0,Y 303.616,Z 383.303,A -85,B 0,C 180,E1 -16111.327,E2 -16111.327} C_VEL
LIN {X 0,Y 303.861,Z 381.748,A -85,B 0,C 180,E1 -16113.979,E2 -16113.979} C_VEL
LIN {X 0,Y 304.02,Z 380.391,A -85,B 0,C 180,E1 -16115.306,E2 -16115.306} C_VEL
LIN {X 0,Y 304.403,Z 377.524,A -85,B 0,C 180,E1 -16117.295,E2 -16117.295} C_VEL
LIN {X 0,Y 304.905,Z 373.638,A -85,B 0,C 180,E1 -16119.285,E2 -16119.285} C_VEL
LIN {X 0,Y 305.714,Z 368.621,A -85,B 0,C 180,E1 -16121.269,E2 -16121.269} C_VEL
LIN {X 0,Y 306.777,Z 362.302,A -85,B 0,C 180,E1 -16123.244,E2 -16123.244} C_VEL
LIN {X 0,Y 308.136,Z 354.391,A -85,B 0,C 180,E1 -16125.206,E2 -16125.206} C_VEL
LIN {X 0,Y 309.8,Z 344.549,A -85,B 0,C 180,E1 -16127.152,E2 -16127.152} C_VEL
LIN {X 0,Y 311.077,Z 335.388,A -85,B 0,C 180,E1 -16128.61,E2 -16128.61} C_VEL
LIN {X 0,Y 312.424,Z 325.405,A -85,B 0,C 180,E1 -16129.892,E2 -16129.892} C_VEL
LIN {X 0,Y 313.357,Z 316.307,A -85,B 0,C 180,E1 -16130.858,E2 -16130.858} C_VEL
LIN {X 0,Y 311.552,Z 305.464,A -85,B 0,C 180,E1 -16131.981,E2 -16131.981} C_VEL
LIN {X 0,Y 308.735,Z 293.206,A -85,B 0,C 180,E1 -16133.049,E2 -16133.049} C_VEL
LIN {X 0,Y 304.738,Z 279.985,A -85,B 0,C 180,E1 -16134.003,E2 -16134.003} C_VEL
LIN {X 0,Y 304.622,Z 279.108,A -85,B 0,C 180,E1 -16134.093,E2 -16134.093} C_VEL
LIN {X 0,Y 304.916,Z 275.566,A -85,B 0,C 180,E1 -16137.451,E2 -16137.451} C_VEL
LIN {X 0,Y 305.167,Z 272.565,A -85,B 0,C 180,E1 -16140.442,E2 -16140.442} C_VEL
LIN {X 0,Y 305.432,Z 269.031,A -85,B 0,C 180,E1 -16144.069,E2 -16144.069} C_VEL
LIN {X 0,Y 305.467,Z 266.559,A -85,B 0,C 180,E1 -16146.741,E2 -16146.741} C_VEL
LIN {X 0,Y 305.404,Z 265.442,A -85,B 0,C 180,E1 -16148.518,E2 -16148.518} C_VEL
LIN {X 0,Y 305.437,Z 265.438,A -85,B 0,C 180,E1 -16152.582,E2 -16152.582} C_VEL
LIN {X 0,Y 305.427,Z 265.441,A -85,B 0,C 180,E1 -16156.345,E2 -16156.345} C_VEL
LIN {X 0,Y 305.46,Z 265.436,A -85,B 0,C 180,E1 -16159.892,E2 -16159.892} C_VEL
LIN {X 0,Y 305.486,Z 265.431,A -85,B 0,C 180,E1 -16163.631,E2 -16163.631} C_VEL
LIN {X 0,Y 305.467,Z 265.434,A -85,B 0,C 180,E1 -16166.483,E2 -16166.483} C_VEL
LIN {X 0,Y 305.466,Z 265.434,A -85,B 0,C 180,E1 -16169.591,E2 -16169.591} C_VEL
LIN {X 0,Y 305.524,Z 265.424,A -85,B 0,C 180,E1 -16172.609,E2 -16172.609} C_VEL
LIN {X 0,Y 305.507,Z 265.432,A -85,B 0,C 180,E1 -16175.539,E2 -16175.539} C_VEL
LIN {X 0,Y 305.498,Z 265.431,A -85,B 0,C 180,E1 -16179.813,E2 -16179.813} C_VEL
LIN {X 0,Y 305.544,Z 265.422,A -85,B 0,C 180,E1 -16182.601,E2 -16182.601} C_VEL
LIN {X 0,Y 305.625,Z 265.416,A -85,B 0,C 180,E1 -16185.387,E2 -16185.387} C_VEL
LIN {X 0,Y 304.919,Z 265.502,A -85,B 0,C 180,E1 -16186.487,E2 -16186.487} C_VEL
LIN {X 0,Y 302.135,Z 265.852,A -85,B 0,C 180,E1 -16188.28,E2 -16188.28} C_VEL
LIN {X 0,Y 299.806,Z 266.146,A -85,B 0,C 180,E1 -16189.735,E2 -16189.735} C_VEL
LIN {X 0,Y 298.802,Z 266.269,A -85,B 0,C 180,E1 -16190.859,E2 -16190.859} C_VEL
LIN {X 0,Y 298.715,Z 266.277,A -85,B 0,C 180,E1 -16191.239,E2 -16191.239} C_VEL
LIN {X 0,Y 298.751,Z 266.272,A -85,B 0,C 180,E1 -16193.245,E2 -16193.245} C_VEL
LIN {X 0,Y 298.907,Z 266.253,A -85,B 0,C 180,E1 -16198.653,E2 -16198.653} C_VEL
LIN {X 0,Y 298.923,Z 266.248,A -85,B 0,C 180,E1 -16201.347,E2 -16201.347} C_VEL
LIN {X 0,Y 298.778,Z 266.268,A -85,B 0,C 180,E1 -16206.754,E2 -16206.754} C_VEL
LIN {X 0,Y 298.627,Z 266.284,A -85,B 0,C 180,E1 -16209.482,E2 -16209.482} C_VEL
LIN {X 0,Y 298.553,Z 266.294,A -85,B 0,C 180,E1 -16213.615,E2 -16213.615} C_VEL
LIN {X 0,Y 298.551,Z 266.297,A -85,B 0,C 180,E1 -16216.409,E2 -16216.409} C_VEL
LIN {X 0,Y 298.512,Z 266.3,A -85,B 0,C 180,E1 -16219.654,E2 -16219.654} C_VEL
LIN {X 0,Y 298.412,Z 266.313,A -85,B 0,C 180,E1 -16223.602,E2 -16223.602} C_VEL
LIN {X 0,Y 298.405,Z 266.313,A -85,B 0,C 180,E1 -16226.583,E2 -16226.583} C_VEL
LIN {X 0,Y 298.395,Z 266.318,A -85,B 0,C 180,E1 -16229.644,E2 -16229.644} C_VEL
LIN {X 0,Y 298.395,Z 266.315,A -85,B 0,C 180,E1 -16232.8,E2 -16232.8} C_VEL
LIN {X 0,Y 298.43,Z 266.312,A -85,B 0,C 180,E1 -16236.803,E2 -16236.803} C_VEL
LIN {X 0,Y 298.375,Z 266.321,A -85,B 0,C 180,E1 -16239.492,E2 -16239.492} C_VEL
LIN {X 0,Y 298.413,Z 266.39,A -85,B 0,C 180,E1 -16243.657,E2 -16243.657} C_VEL
LIN {X 0,Y 299.064,Z 270.002,A -85,B 0,C 180,E1 -16247.039,E2 -16247.039} C_VEL
LIN {X 0,Y 299.761,Z 274.247,A -85,B 0,C 180,E1 -16250.726,E2 -16250.726} C_VEL
LIN {X 0,Y 299.999,Z 276.774,A -85,B 0,C 180,E1 -16252.798,E2 -16252.798} C_VEL
LIN {X 0,Y 300.005,Z 279.663,A -85,B 0,C 180,E1 -16255.077,E2 -16255.077} C_VEL
LIN {X 0,Y 299.184,Z 284.748,A -85,B 0,C 180,E1 -16258.882,E2 -16258.882} C_VEL
LIN {X 0,Y 298.319,Z 290.974,A -85,B 0,C 180,E1 -16263.409,E2 -16263.409} C_VEL
LIN {X 0,Y 298,Z 293.855,A -85,B 0,C 180,E1 -16265.412,E2 -16265.412} C_VEL
LIN {X 0,Y 301.245,Z 307.281,A -85,B 0,C 180,E1 -16266.289,E2 -16266.289} C_VEL
LIN {X 0,Y 303.494,Z 319.958,A -85,B 0,C 180,E1 -16267.329,E2 -16267.329} C_VEL
LIN {X 0,Y 304.904,Z 332.079,A -85,B 0,C 180,E1 -16268.536,E2 -16268.536} C_VEL
LIN {X 0,Y 305.176,Z 339.92,A -85,B 0,C 180,E1 -16269.439,E2 -16269.439} C_VEL
LIN {X 0,Y 303.408,Z 351.45,A -85,B 0,C 180,E1 -16270.902,E2 -16270.902} C_VEL
LIN {X 0,Y 301.936,Z 360.74,A -85,B 0,C 180,E1 -16272.386,E2 -16272.386} C_VEL
LIN {X 0,Y 300.586,Z 369.214,A -85,B 0,C 180,E1 -16274.054,E2 -16274.054} C_VEL
LIN {X 0,Y 299.234,Z 377.488,A -85,B 0,C 180,E1 -16276.07,E2 -16276.07} C_VEL
LIN {X 0,Y 298.09,Z 384.157,A -85,B 0,C 180,E1 -16278.094,E2 -16278.094} C_VEL
LIN {X 0,Y 297.255,Z 390.263,A -85,B 0,C 180,E1 -16280.473,E2 -16280.473} C_VEL
LIN {X 0,Y 296.79,Z 394.233,A -85,B 0,C 180,E1 -16282.516,E2 -16282.516} C_VEL
LIN {X 0,Y 296.552,Z 397.168,A -85,B 0,C 180,E1 -16284.56,E2 -16284.56} C_VEL
LIN {X 0,Y 296.529,Z 398.566,A -85,B 0,C 180,E1 -16285.923,E2 -16285.923} C_VEL
LIN {X 0,Y 296.533,Z 399.564,A -85,B 0,C 180,E1 -16287.283,E2 -16287.283} C_VEL
LIN {X 0,Y 296.493,Z 400.171,A -85,B 0,C 180,E1 -16288.642,E2 -16288.642} C_VEL
LIN {X 0,Y 296.519,Z 400.386,A -85,B 0,C 180,E1 -16290,E2 -16290} C_VEL
LIN {X 0,Y 296.493,Z 400.164,A -85,B 0,C 180,E1 -16291.358,E2 -16291.358} C_VEL
LIN {X 0,Y 296.531,Z 399.553,A -85,B 0,C 180,E1 -16292.717,E2 -16292.717} C_VEL
LIN {X 0,Y 296.505,Z 398.55,A -85,B 0,C 180,E1 -16294.078,E2 -16294.078} C_VEL
LIN {X 0,Y 296.546,Z 397.06,A -85,B 0,C 180,E1 -16295.508,E2 -16295.508} C_VEL
LIN {X 0,Y 296.899,Z 392.967,A -85,B 0,C 180,E1 -16298.165,E2 -16298.165} C_VEL
LIN {X 0,Y 297.443,Z 388.616,A -85,B 0,C 180,E1 -16300.207,E2 -16300.207} C_VEL
LIN {X 0,Y 298.216,Z 383.076,A -85,B 0,C 180,E1 -16302.245,E2 -16302.245} C_VEL
LIN {X 0,Y 299.449,Z 376.169,A -85,B 0,C 180,E1 -16304.266,E2 -16304.266} C_VEL
LIN {X 0,Y 300.918,Z 367.524,A -85,B 0,C 180,E1 -16306.276,E2 -16306.276} C_VEL
LIN {X 0,Y 302.253,Z 358.659,A -85,B 0,C 180,E1 -16307.944,E2 -16307.944} C_VEL
LIN {X 0,Y 303.953,Z 347.755,A -85,B 0,C 180,E1 -16309.589,E2 -16309.589} C_VEL
LIN {X 0,Y 305.225,Z 338.291,A -85,B 0,C 180,E1 -16310.733,E2 -16310.733} C_VEL
LIN {X 0,Y 304.424,Z 327.4,A -85,B 0,C 180,E1 -16311.937,E2 -16311.937} C_VEL
LIN {X 0,Y 302.657,Z 314.69,A -85,B 0,C 180,E1 -16313.101,E2 -16313.101} C_VEL
LIN {X 0,Y 300.108,Z 302.36,A -85,B 0,C 180,E1 -16314.033,E2 -16314.033} C_VEL
LIN {X 0,Y 297.996,Z 293.753,A -85,B 0,C 180,E1 -16314.573,E2 -16314.573} C_VEL
LIN {X 0,Y 298.592,Z 288.878,A -85,B 0,C 180,E1 -16318.082,E2 -16318.082} C_VEL
LIN {X 0,Y 299.418,Z 283.068,A -85,B 0,C 180,E1 -16322.328,E2 -16322.328} C_VEL
LIN {X 0,Y 299.98,Z 279.628,A -85,B 0,C 180,E1 -16324.916,E2 -16324.916} C_VEL
LIN {X 0,Y 299.878,Z 275.269,A -85,B 0,C 180,E1 -16328.393,E2 -16328.393} C_VEL
LIN {X 0,Y 299.351,Z 271.834,A -85,B 0,C 180,E1 -16331.299,E2 -16331.299} C_VEL
LIN {X 0,Y 298.623,Z 267.671,A -85,B 0,C 180,E1 -16335.086,E2 -16335.086} C_VEL
LIN {X 0,Y 298.388,Z 266.318,A -85,B 0,C 180,E1 -16336.455,E2 -16336.455} C_VEL
LIN {X 0,Y 298.385,Z 266.318,A -85,B 0,C 180,E1 -16341.011,E2 -16341.011} C_VEL
LIN {X 0,Y 298.406,Z 266.314,A -85,B 0,C 180,E1 -16343.928,E2 -16343.928} C_VEL
LIN {X 0,Y 298.394,Z 266.316,A -85,B 0,C 180,E1 -16347.2,E2 -16347.2} C_VEL
LIN {X 0,Y 298.403,Z 266.316,A -85,B 0,C 180,E1 -16350.625,E2 -16350.625} C_VEL
LIN {X 0,Y 298.424,Z 266.311,A -85,B 0,C 180,E1 -16354.918,E2 -16354.918} C_VEL
LIN {X 0,Y 298.434,Z 266.31,A -85,B 0,C 180,E1 -16359.314,E2 -16359.314} C_VEL
LIN {X 0,Y 298.536,Z 266.298,A -85,B 0,C 180,E1 -16362.179,E2 -16362.179} C_VEL
LIN {X 0,Y 298.595,Z 266.289,A -85,B 0,C 180,E1 -16364.995,E2 -16364.995} C_VEL
LIN {X 0,Y 298.584,Z 266.291,A -85,B 0,C 180,E1 -16369.146,E2 -16369.146} C_VEL
LIN {X 0,Y 298.719,Z 266.275,A -85,B 0,C 180,E1 -16371.885,E2 -16371.885} C_VEL
LIN {X 0,Y 298.655,Z 266.281,A -85,B 0,C 180,E1 -16374.599,E2 -16374.599} C_VEL
LIN {X 0,Y 298.923,Z 266.247,A -85,B 0,C 180,E1 -16378.653,E2 -16378.653} C_VEL
LIN {X 0,Y 298.915,Z 266.251,A -85,B 0,C 180,E1 -16381.347,E2 -16381.347} C_VEL
LIN {X 0,Y 298.765,Z 266.27,A -85,B 0,C 180,E1 -16386.755,E2 -16386.755} C_VEL
LIN {X 0,Y 298.627,Z 266.285,A -85,B 0,C 180,E1 -16389.482,E2 -16389.482} C_VEL
LIN {X 0,Y 298.547,Z 266.295,A -85,B 0,C 180,E1 -16393.616,E2 -16393.616} C_VEL
LIN {X 0,Y 298.488,Z 266.304,A -85,B 0,C 180,E1 -16396.412,E2 -16396.412} C_VEL
LIN {X 0,Y 298.484,Z 266.302,A -85,B 0,C 180,E1 -16399.639,E2 -16399.639} C_VEL
LIN {X 0,Y 298.43,Z 266.309,A -85,B 0,C 180,E1 -16403.6,E2 -16403.6} C_VEL
LIN {X 0,Y 298.491,Z 266.304,A -85,B 0,C 180,E1 -16406.574,E2 -16406.574} C_VEL
LIN {X 0,Y 298.425,Z 266.31,A -85,B 0,C 180,E1 -16409.641,E2 -16409.641} C_VEL
LIN {X 0,Y 298.397,Z 266.314,A -85,B 0,C 180,E1 -16412.8,E2 -16412.8} C_VEL
LIN {X 0,Y 298.447,Z 266.307,A -85,B 0,C 180,E1 -16416.808,E2 -16416.808} C_VEL
LIN {X 0,Y 298.409,Z 266.314,A -85,B 0,C 180,E1 -16419.486,E2 -16419.486} C_VEL
LIN {X 0,Y 298.4,Z 266.313,A -85,B 0,C 180,E1 -16423.103,E2 -16423.103} C_VEL
LIN {X 0,Y 298.371,Z 266.317,A -85,B 0,C 180,E1 -16426.915,E2 -16426.915} C_VEL
LIN {X 0,Y 298.346,Z 266.323,A -85,B 0,C 180,E1 -16431.02,E2 -16431.02} C_VEL
LIN {X 0,Y 298.374,Z 266.625,A -85,B 0,C 180,E1 -16432.236,E2 -16432.236} C_VEL
